Yaskawa INFORM job: A_ROOF_UPPER_0614_2_PAINT_18.JBI

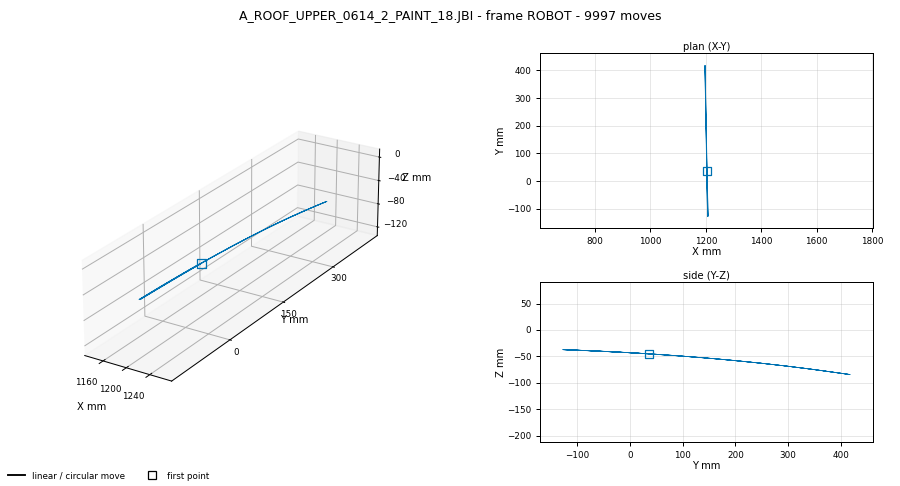
[picture p0: tool path of A_ROOF_UPPER_0614_2_PAINT_18.JBI in frame ROBOT, 9997 of 9997 moves have a stored position in this frame; points joined in program order, loops and branches not executed]
/JOB
//NAME A_ROOF_UPPER_0614_2_PAINT18
//POS
///NPOS 9997,0,0,0,0,0
///TOOL 1
///USER 0
///POSTYPE ROBOT
///RECTAN
///RCONF 1,0,0,0,0,0,0,0,0,0,0,0,0,0,0,0,0,0,0,0,0,0,0,0
C00000=1205.007,36.584,-45.184,-179.345,5.640,148.798
C00001=1205.012,36.335,-45.168,-179.348,5.639,148.799
C00002=1205.017,36.086,-45.153,-179.350,5.639,148.800
C00003=1205.023,35.836,-45.137,-179.353,5.638,148.800
C00004=1205.027,35.586,-45.122,-179.356,5.638,148.801
C00005=1205.032,35.337,-45.106,-179.358,5.637,148.801
C00006=1205.037,35.088,-45.090,-179.360,5.636,148.802
C00007=1205.042,34.839,-45.075,-179.363,5.636,148.803
C00008=1205.047,34.589,-45.059,-179.366,5.635,148.803
C00009=1205.052,34.340,-45.043,-179.368,5.635,148.804
C00010=1205.057,34.090,-45.028,-179.371,5.634,148.805
C00011=1205.062,33.841,-45.013,-179.373,5.633,148.805
C00012=1205.067,33.591,-44.997,-179.376,5.633,148.806
C00013=1205.072,33.342,-44.982,-179.378,5.632,148.807
C00014=1205.077,33.093,-44.966,-179.381,5.632,148.807
C00015=1205.082,32.843,-44.951,-179.383,5.631,148.808
C00016=1205.086,32.593,-44.935,-179.386,5.630,148.808
C00017=1205.092,32.344,-44.920,-179.389,5.630,148.809
C00018=1205.097,32.094,-44.905,-179.391,5.629,148.810
C00019=1205.102,31.845,-44.890,-179.394,5.629,148.810
C00020=1205.107,31.595,-44.874,-179.396,5.628,148.811
C00021=1205.112,31.345,-44.858,-179.399,5.627,148.811
C00022=1205.117,31.096,-44.843,-179.401,5.627,148.812
C00023=1205.122,30.847,-44.828,-179.404,5.626,148.813
C00024=1205.127,30.598,-44.813,-179.407,5.626,148.814
C00025=1205.132,30.348,-44.797,-179.409,5.625,148.814
C00026=1205.137,30.098,-44.781,-179.411,5.624,148.815
C00027=1205.142,29.849,-44.766,-179.414,5.624,148.815
C00028=1205.147,29.600,-44.750,-179.417,5.623,148.816
C00029=1205.152,29.331,-44.735,-179.419,5.623,148.817
C00030=1205.158,29.062,-44.718,-179.422,5.622,148.817
C00031=1205.164,28.793,-44.701,-179.425,5.622,148.818
C00032=1205.169,28.525,-44.686,-179.427,5.621,148.819
C00033=1205.174,28.274,-44.670,-179.430,5.621,148.819
C00034=1205.178,28.025,-44.655,-179.432,5.620,148.820
C00035=1205.184,27.776,-44.639,-179.435,5.619,148.821
C00036=1205.188,27.527,-44.624,-179.437,5.619,148.821
C00037=1205.194,27.277,-44.609,-179.440,5.618,148.822
C00038=1205.199,27.028,-44.594,-179.443,5.618,148.823
C00039=1205.204,26.778,-44.579,-179.445,5.617,148.823
C00040=1205.208,26.529,-44.563,-179.447,5.616,148.824
C00041=1205.213,26.279,-44.548,-179.450,5.616,148.824
C00042=1205.218,26.029,-44.534,-179.453,5.615,148.825
C00043=1205.224,25.780,-44.518,-179.455,5.615,148.826
C00044=1205.228,25.531,-44.503,-179.458,5.614,148.826
C00045=1205.234,25.282,-44.487,-179.460,5.613,148.827
C00046=1205.239,25.032,-44.473,-179.463,5.613,148.828
C00047=1205.244,24.782,-44.457,-179.465,5.612,148.828
C00048=1205.248,24.533,-44.442,-179.468,5.612,148.829
C00049=1205.253,24.283,-44.428,-179.471,5.611,148.830
C00050=1205.259,24.034,-44.412,-179.473,5.610,148.830
C00051=1205.263,23.784,-44.397,-179.476,5.610,148.831
C00052=1205.269,23.534,-44.382,-179.478,5.609,148.831
C00053=1205.274,23.285,-44.367,-179.481,5.609,148.832
C00054=1205.279,23.036,-44.352,-179.483,5.608,148.833
C00055=1205.284,22.786,-44.338,-179.486,5.608,148.833
C00056=1205.289,22.537,-44.323,-179.488,5.607,148.834
C00057=1205.294,22.288,-44.307,-179.490,5.607,148.835
C00058=1205.299,22.038,-44.293,-179.493,5.607,148.835
C00059=1205.304,21.789,-44.277,-179.496,5.606,148.836
C00060=1205.309,21.538,-44.262,-179.498,5.606,148.837
C00061=1205.313,21.289,-44.247,-179.501,5.605,148.837
C00062=1205.319,21.040,-44.232,-179.503,5.604,148.838
C00063=1205.324,20.790,-44.218,-179.506,5.604,148.838
C00064=1205.328,20.541,-44.203,-179.508,5.603,148.839
C00065=1205.334,20.291,-44.188,-179.511,5.603,148.840
C00066=1205.339,20.042,-44.173,-179.514,5.602,148.840
C00067=1205.344,19.792,-44.158,-179.516,5.601,148.841
C00068=1205.349,19.543,-44.143,-179.519,5.601,148.842
C00069=1205.354,19.293,-44.129,-179.521,5.600,148.842
C00070=1205.359,19.044,-44.114,-179.524,5.600,148.843
C00071=1205.364,18.794,-44.099,-179.526,5.599,148.844
C00072=1205.369,18.545,-44.084,-179.529,5.599,148.844
C00073=1205.374,18.295,-44.069,-179.531,5.599,148.845
C00074=1205.379,18.046,-44.054,-179.533,5.598,148.845
C00075=1205.384,17.796,-44.040,-179.536,5.598,148.846
C00076=1205.389,17.547,-44.025,-179.539,5.597,148.847
C00077=1205.395,17.297,-44.010,-179.541,5.597,148.847
C00078=1205.399,17.048,-43.995,-179.544,5.596,148.848
C00079=1205.404,16.798,-43.980,-179.546,5.595,148.849
C00080=1205.409,16.549,-43.965,-179.549,5.595,148.849
C00081=1205.414,16.299,-43.951,-179.551,5.594,148.850
C00082=1205.419,16.049,-43.936,-179.554,5.594,148.851
C00083=1205.424,15.800,-43.921,-179.557,5.593,148.851
C00084=1205.429,15.550,-43.907,-179.559,5.593,148.852
C00085=1205.434,15.301,-43.891,-179.561,5.592,148.852
C00086=1205.439,15.051,-43.877,-179.564,5.592,148.853
C00087=1205.444,14.802,-43.863,-179.566,5.592,148.854
C00088=1205.449,14.552,-43.848,-179.569,5.591,148.855
C00089=1205.455,14.302,-43.833,-179.571,5.591,148.855
C00090=1205.460,14.053,-43.819,-179.574,5.590,148.856
C00091=1205.464,13.804,-43.804,-179.576,5.589,148.856
C00092=1205.469,13.554,-43.789,-179.579,5.589,148.857
C00093=1205.475,13.305,-43.776,-179.582,5.588,148.858
C00094=1205.480,13.056,-43.760,-179.584,5.588,148.858
C00095=1205.485,12.806,-43.746,-179.587,5.587,148.859
C00096=1205.490,12.556,-43.731,-179.589,5.588,148.860
C00097=1205.495,12.307,-43.716,-179.592,5.587,148.860
C00098=1205.500,12.057,-43.702,-179.594,5.586,148.861
C00099=1205.505,11.808,-43.688,-179.596,5.586,148.862
C00100=1205.510,11.558,-43.672,-179.599,5.585,148.862
C00101=1205.515,11.308,-43.658,-179.602,5.585,148.863
C00102=1205.520,11.059,-43.644,-179.604,5.584,148.864
C00103=1205.525,10.809,-43.629,-179.607,5.584,148.864
C00104=1205.530,10.561,-43.615,-179.609,5.583,148.865
C00105=1205.535,10.311,-43.601,-179.612,5.582,148.865
C00106=1205.540,10.061,-43.586,-179.614,5.583,148.866
C00107=1205.545,9.812,-43.572,-179.617,5.582,148.867
C00108=1205.551,9.562,-43.557,-179.619,5.582,148.868
C00109=1205.555,9.312,-43.542,-179.622,5.581,148.868
C00110=1205.560,9.063,-43.528,-179.624,5.580,148.869
C00111=1205.565,8.813,-43.514,-179.627,5.580,148.869
C00112=1205.570,8.563,-43.499,-179.629,5.579,148.870
C00113=1205.576,8.314,-43.485,-179.632,5.579,148.871
C00114=1205.581,8.065,-43.471,-179.635,5.578,148.871
C00115=1205.585,7.815,-43.456,-179.637,5.578,148.872
C00116=1205.590,7.566,-43.442,-179.639,5.578,148.873
C00117=1205.595,7.316,-43.428,-179.642,5.577,148.873
C00118=1205.600,7.066,-43.413,-179.644,5.577,148.874
C00119=1205.606,6.817,-43.399,-179.647,5.576,148.875
C00120=1205.611,6.568,-43.385,-179.649,5.576,148.875
C00121=1205.616,6.318,-43.371,-179.652,5.575,148.876
C00122=1205.621,6.068,-43.357,-179.655,5.575,148.877
C00123=1205.625,5.819,-43.342,-179.657,5.575,148.877
C00124=1205.630,5.569,-43.327,-179.659,5.574,148.878
C00125=1205.636,5.320,-43.313,-179.662,5.573,148.879
C00126=1205.641,5.071,-43.299,-179.664,5.573,148.879
C00127=1205.646,4.821,-43.285,-179.667,5.572,148.880
C00128=1205.651,4.571,-43.271,-179.670,5.572,148.881
C00129=1205.656,4.322,-43.256,-179.672,5.571,148.881
C00130=1205.661,4.073,-43.242,-179.675,5.571,148.882
C00131=1205.666,3.823,-43.228,-179.677,5.571,148.882
C00132=1205.671,3.573,-43.214,-179.679,5.570,148.883
C00133=1205.677,3.304,-43.199,-179.682,5.570,148.884
C00134=1205.682,3.035,-43.183,-179.684,5.569,148.884
C00135=1205.687,2.766,-43.168,-179.687,5.569,148.885
C00136=1205.694,2.497,-43.152,-179.690,5.569,148.886
C00137=1205.698,2.248,-43.139,-179.692,5.568,148.887
C00138=1205.703,1.998,-43.124,-179.695,5.567,148.887
C00139=1205.708,1.748,-43.110,-179.698,5.567,148.888
C00140=1205.714,1.499,-43.097,-179.700,5.566,148.889
C00141=1205.718,1.249,-43.082,-179.703,5.566,148.889
C00142=1205.723,0.999,-43.068,-179.705,5.566,148.890
C00143=1205.728,0.750,-43.054,-179.708,5.566,148.891
C00144=1205.734,0.501,-43.040,-179.710,5.565,148.891
C00145=1205.739,0.251,-43.026,-179.713,5.564,148.892
C00146=1205.744,0.001,-43.011,-179.715,5.564,148.893
C00147=1205.749,-0.249,-42.997,-179.718,5.563,148.893
C00148=1205.754,-0.497,-42.984,-179.720,5.564,148.894
C00149=1205.759,-0.747,-42.970,-179.723,5.563,148.895
C00150=1205.764,-0.997,-42.956,-179.725,5.563,148.895
C00151=1205.769,-1.247,-42.942,-179.727,5.562,148.896
C00152=1205.774,-1.496,-42.928,-179.730,5.561,148.896
C00153=1205.779,-1.746,-42.914,-179.733,5.561,148.897
C00154=1205.784,-1.995,-42.899,-179.735,5.561,148.898
C00155=1205.789,-2.244,-42.886,-179.737,5.561,148.898
C00156=1205.794,-2.494,-42.872,-179.740,5.560,148.899
C00157=1205.799,-2.744,-42.858,-179.743,5.560,148.900
C00158=1205.805,-2.993,-42.844,-179.745,5.559,148.901
C00159=1205.810,-3.243,-42.830,-179.748,5.558,148.901
C00160=1205.815,-3.493,-42.816,-179.750,5.559,148.902
C00161=1205.820,-3.742,-42.803,-179.752,5.558,148.902
C00162=1205.825,-3.992,-42.789,-179.755,5.558,148.903
C00163=1205.830,-4.241,-42.775,-179.758,5.557,148.904
C00164=1205.835,-4.491,-42.760,-179.760,5.557,148.904
C00165=1205.840,-4.740,-42.746,-179.763,5.556,148.905
C00166=1205.845,-4.990,-42.733,-179.765,5.556,148.906
C00167=1205.850,-5.239,-42.719,-179.767,5.556,148.906
C00168=1205.855,-5.489,-42.705,-179.770,5.555,148.907
C00169=1205.861,-5.739,-42.692,-179.772,5.555,148.908
C00170=1205.865,-5.988,-42.678,-179.775,5.554,148.908
C00171=1205.870,-6.238,-42.664,-179.778,5.554,148.909
C00172=1205.875,-6.487,-42.650,-179.780,5.554,148.910
C00173=1205.881,-6.737,-42.637,-179.783,5.553,148.910
C00174=1205.885,-6.986,-42.623,-179.785,5.552,148.911
C00175=1205.890,-7.236,-42.609,-179.787,5.552,148.912
C00176=1205.896,-7.486,-42.595,-179.790,5.552,148.912
C00177=1205.900,-7.735,-42.582,-179.792,5.552,148.913
C00178=1205.905,-7.985,-42.567,-179.795,5.551,148.914
C00179=1205.911,-8.234,-42.554,-179.797,5.551,148.914
C00180=1205.916,-8.484,-42.540,-179.800,5.550,148.915
C00181=1205.921,-8.733,-42.527,-179.803,5.550,148.916
C00182=1205.926,-8.983,-42.513,-179.805,5.549,148.916
C00183=1205.931,-9.233,-42.499,-179.807,5.549,148.917
C00184=1205.936,-9.482,-42.486,-179.810,5.549,148.918
C00185=1205.941,-9.732,-42.472,-179.812,5.548,148.918
C00186=1205.947,-9.982,-42.459,-179.815,5.548,148.919
C00187=1205.951,-10.231,-42.445,-179.818,5.547,148.920
C00188=1205.956,-10.481,-42.431,-179.820,5.548,148.920
C00189=1205.962,-10.730,-42.418,-179.822,5.547,148.921
C00190=1205.966,-10.980,-42.404,-179.824,5.546,148.922
C00191=1205.972,-11.229,-42.391,-179.827,5.546,148.922
C00192=1205.977,-11.479,-42.377,-179.830,5.545,148.923
C00193=1205.982,-11.728,-42.364,-179.832,5.546,148.924
C00194=1205.987,-11.978,-42.350,-179.835,5.545,148.924
C00195=1205.992,-12.228,-42.337,-179.837,5.545,148.925
C00196=1205.997,-12.477,-42.323,-179.840,5.544,148.926
C00197=1206.002,-12.727,-42.310,-179.842,5.544,148.926
C00198=1206.007,-12.976,-42.296,-179.844,5.544,148.927
C00199=1206.013,-13.226,-42.282,-179.847,5.543,148.928
C00200=1206.018,-13.475,-42.269,-179.849,5.543,148.928
C00201=1206.023,-13.725,-42.255,-179.852,5.542,148.929
C00202=1206.028,-13.974,-42.242,-179.854,5.543,148.930
C00203=1206.033,-14.224,-42.228,-179.857,5.542,148.930
C00204=1206.038,-14.473,-42.215,-179.859,5.542,148.931
C00205=1206.043,-14.723,-42.202,-179.862,5.541,148.932
C00206=1206.049,-14.973,-42.188,-179.864,5.540,148.932
C00207=1206.053,-15.223,-42.175,-179.866,5.541,148.933
C00208=1206.059,-15.472,-42.162,-179.869,5.540,148.934
C00209=1206.063,-15.722,-42.148,-179.872,5.540,148.934
C00210=1206.069,-15.971,-42.135,-179.874,5.539,148.935
C00211=1206.073,-16.221,-42.121,-179.877,5.539,148.936
C00212=1206.079,-16.470,-42.108,-179.879,5.539,148.936
C00213=1206.084,-16.720,-42.095,-179.882,5.538,148.937
C00214=1206.089,-16.969,-42.081,-179.884,5.538,148.937
C00215=1206.094,-17.219,-42.068,-179.887,5.537,148.938
C00216=1206.100,-17.469,-42.055,-179.889,5.537,148.939
C00217=1206.104,-17.718,-42.041,-179.891,5.537,148.940
C00218=1206.110,-17.968,-42.028,-179.894,5.536,148.940
C00219=1206.114,-18.218,-42.015,-179.897,5.536,148.941
C00220=1206.120,-18.467,-42.001,-179.899,5.536,148.942
C00221=1206.124,-18.717,-41.988,-179.901,5.536,148.942
C00222=1206.130,-18.967,-41.975,-179.903,5.535,148.943
C00223=1206.134,-19.216,-41.961,-179.906,5.534,148.943
C00224=1206.140,-19.466,-41.948,-179.909,5.534,148.944
C00225=1206.145,-19.715,-41.935,-179.911,5.534,148.945
C00226=1206.151,-19.965,-41.922,-179.914,5.534,148.946
C00227=1206.155,-20.214,-41.908,-179.916,5.533,148.946
C00228=1206.161,-20.464,-41.895,-179.919,5.533,148.947
C00229=1206.166,-20.714,-41.882,-179.921,5.533,148.948
C00230=1206.170,-20.964,-41.869,-179.923,5.532,148.948
C00231=1206.176,-21.213,-41.855,-179.926,5.532,148.949
C00232=1206.181,-21.462,-41.843,-179.928,5.531,148.950
C00233=1206.186,-21.712,-41.829,-179.930,5.532,148.950
C00234=1206.191,-21.962,-41.817,-179.933,5.531,148.951
C00235=1206.196,-22.212,-41.804,-179.936,5.531,148.952
C00236=1206.201,-22.461,-41.790,-179.938,5.530,148.952
C00237=1206.206,-22.730,-41.776,-179.941,5.530,148.953
C00238=1206.212,-23.000,-41.762,-179.943,5.530,148.954
C00239=1206.218,-23.269,-41.747,-179.946,5.530,148.954
C00240=1206.223,-23.539,-41.733,-179.949,5.529,148.955
C00241=1206.229,-23.788,-41.720,-179.951,5.529,148.956
C00242=1206.234,-24.038,-41.707,-179.954,5.528,148.956
C00243=1206.239,-24.288,-41.695,-179.956,5.528,148.957
C00244=1206.244,-24.537,-41.681,-179.959,5.528,148.958
C00245=1206.249,-24.787,-41.668,-179.961,5.528,148.959
C00246=1206.254,-25.036,-41.655,-179.963,5.527,148.959
C00247=1206.259,-25.286,-41.642,-179.966,5.527,148.960
C00248=1206.264,-25.536,-41.629,-179.968,5.527,148.960
C00249=1206.269,-25.785,-41.616,-179.971,5.526,148.961
C00250=1206.274,-26.035,-41.604,-179.973,5.526,148.962
C00251=1206.280,-26.285,-41.590,-179.976,5.526,148.963
C00252=1206.285,-26.534,-41.578,-179.978,5.525,148.963
C00253=1206.289,-26.784,-41.565,-179.981,5.525,148.964
C00254=1206.295,-27.034,-41.552,-179.984,5.524,148.965
C00255=1206.300,-27.283,-41.539,-179.985,5.524,148.965
C00256=1206.305,-27.532,-41.525,-179.988,5.524,148.966
C00257=1206.310,-27.782,-41.513,-179.990,5.523,148.966
C00258=1206.316,-28.031,-41.499,-179.993,5.523,148.967
C00259=1206.320,-28.281,-41.487,-179.995,5.523,148.968
C00260=1206.325,-28.531,-41.474,-179.998,5.523,148.969
C00261=1206.331,-28.780,-41.461,179.999,5.522,148.969
C00262=1206.336,-29.030,-41.448,179.997,5.523,148.970
C00263=1206.341,-29.280,-41.435,179.995,5.522,148.970
C00264=1206.346,-29.529,-41.423,179.993,5.521,148.971
C00265=1206.350,-29.779,-41.410,179.990,5.521,148.972
C00266=1206.356,-30.029,-41.396,179.988,5.521,148.973
C00267=1206.361,-30.278,-41.384,179.985,5.521,148.973
C00268=1206.366,-30.529,-41.372,179.982,5.520,148.974
C00269=1206.371,-30.778,-41.359,179.980,5.520,148.975
C00270=1206.377,-31.028,-41.346,179.978,5.520,148.975
C00271=1206.382,-31.277,-41.333,179.975,5.520,148.976
C00272=1206.387,-31.527,-41.320,179.973,5.519,148.976
C00273=1206.392,-31.776,-41.308,179.971,5.519,148.977
C00274=1206.397,-32.026,-41.295,179.968,5.519,148.978
C00275=1206.402,-32.275,-41.282,179.966,5.518,148.979
C00276=1206.408,-32.525,-41.269,179.963,5.518,148.979
C00277=1206.413,-32.774,-41.256,179.961,5.518,148.980
C00278=1206.418,-33.024,-41.244,179.958,5.518,148.981
C00279=1206.423,-33.274,-41.232,179.955,5.517,148.981
C00280=1206.428,-33.524,-41.219,179.954,5.517,148.982
C00281=1206.433,-33.773,-41.206,179.951,5.517,148.983
C00282=1206.439,-34.023,-41.193,179.949,5.516,148.983
C00283=1206.444,-34.272,-41.180,179.946,5.516,148.984
C00284=1206.448,-34.522,-41.167,179.944,5.516,148.985
C00285=1206.454,-34.772,-41.156,179.941,5.516,148.985
C00286=1206.459,-35.021,-41.143,179.938,5.515,148.986
C00287=1206.464,-35.271,-41.130,179.936,5.515,148.987
C00288=1206.469,-35.521,-41.117,179.934,5.515,148.987
C00289=1206.474,-35.770,-41.105,179.932,5.514,148.988
C00290=1206.480,-36.020,-41.092,179.929,5.514,148.989
C00291=1206.485,-36.270,-41.080,179.927,5.514,148.989
C00292=1206.490,-36.519,-41.067,179.924,5.514,148.990
C00293=1206.495,-36.769,-41.054,179.921,5.513,148.991
C00294=1206.500,-37.018,-41.041,179.919,5.513,148.991
C00295=1206.505,-37.268,-41.030,179.917,5.513,148.992
C00296=1206.510,-37.517,-41.017,179.914,5.512,148.993
C00297=1206.515,-37.767,-41.004,179.913,5.512,148.993
C00298=1206.520,-38.017,-40.992,179.910,5.512,148.994
C00299=1206.525,-38.267,-40.980,179.907,5.511,148.995
C00300=1206.530,-38.516,-40.967,179.905,5.512,148.995
C00301=1206.536,-38.765,-40.954,179.902,5.511,148.996
C00302=1206.541,-39.015,-40.942,179.900,5.511,148.997
C00303=1206.546,-39.265,-40.930,179.897,5.510,148.997
C00304=1206.551,-39.515,-40.917,179.895,5.511,148.998
C00305=1206.556,-39.765,-40.905,179.892,5.510,148.999
C00306=1206.561,-40.014,-40.892,179.890,5.509,148.999
C00307=1206.566,-40.263,-40.880,179.888,5.510,149.000
C00308=1206.572,-40.513,-40.868,179.885,5.509,149.001
C00309=1206.577,-40.762,-40.855,179.883,5.509,149.001
C00310=1206.582,-41.012,-40.843,179.881,5.509,149.002
C00311=1206.587,-41.262,-40.830,179.878,5.509,149.003
C00312=1206.592,-41.512,-40.818,179.875,5.508,149.004
C00313=1206.597,-41.762,-40.806,179.873,5.509,149.004
C00314=1206.603,-42.011,-40.793,179.871,5.508,149.005
C00315=1206.608,-42.260,-40.781,179.868,5.507,149.005
C00316=1206.613,-42.510,-40.769,179.866,5.508,149.006
C00317=1206.618,-42.760,-40.756,179.864,5.507,149.007
C00318=1206.624,-43.009,-40.744,179.861,5.507,149.008
C00319=1206.628,-43.259,-40.731,179.859,5.507,149.008
C00320=1206.633,-43.509,-40.719,179.856,5.507,149.009
C00321=1206.639,-43.759,-40.707,179.854,5.506,149.010
C00322=1206.644,-44.008,-40.694,179.852,5.506,149.010
C00323=1206.649,-44.258,-40.682,179.849,5.506,149.011
C00324=1206.654,-44.507,-40.670,179.847,5.505,149.011
C00325=1206.660,-44.757,-40.658,179.845,5.506,149.012
C00326=1206.665,-45.007,-40.645,179.842,5.505,149.013
C00327=1206.670,-45.256,-40.634,179.839,5.505,149.014
C00328=1206.675,-45.505,-40.621,179.837,5.504,149.014
C00329=1206.680,-45.755,-40.610,179.835,5.505,149.015
C00330=1206.685,-46.005,-40.597,179.832,5.504,149.015
C00331=1206.690,-46.255,-40.585,179.830,5.503,149.016
C00332=1206.695,-46.505,-40.572,179.828,5.504,149.017
C00333=1206.701,-46.755,-40.560,179.825,5.503,149.018
C00334=1206.706,-47.004,-40.548,179.822,5.503,149.018
C00335=1206.711,-47.254,-40.536,179.820,5.503,149.019
C00336=1206.716,-47.503,-40.524,179.818,5.503,149.020
C00337=1206.721,-47.753,-40.512,179.815,5.503,149.020
C00338=1206.727,-48.003,-40.500,179.813,5.502,149.021
C00339=1206.732,-48.252,-40.487,179.811,5.502,149.022
C00340=1206.737,-48.502,-40.476,179.809,5.502,149.022
C00341=1206.742,-48.772,-40.463,179.806,5.501,149.023
C00342=1206.748,-49.041,-40.449,179.803,5.501,149.024
C00343=1206.753,-49.312,-40.436,179.800,5.501,149.025
C00344=1206.759,-49.582,-40.423,179.797,5.500,149.025
C00345=1206.764,-49.832,-40.411,179.795,5.501,149.026
C00346=1206.769,-50.081,-40.399,179.793,5.500,149.026
C00347=1206.775,-50.331,-40.387,179.790,5.500,149.027
C00348=1206.780,-50.581,-40.375,179.788,5.500,149.028
C00349=1206.784,-50.830,-40.363,179.786,5.499,149.029
C00350=1206.790,-51.080,-40.351,179.783,5.499,149.029
C00351=1206.795,-51.330,-40.339,179.781,5.499,149.030
C00352=1206.800,-51.579,-40.327,179.778,5.499,149.031
C00353=1206.805,-51.829,-40.315,179.777,5.499,149.031
C00354=1206.810,-52.079,-40.304,179.774,5.498,149.032
C00355=1206.816,-52.328,-40.291,179.771,5.498,149.033
C00356=1206.821,-52.578,-40.279,179.769,5.498,149.033
C00357=1206.826,-52.828,-40.268,179.767,5.498,149.034
C00358=1206.831,-53.077,-40.255,179.764,5.497,149.035
C00359=1206.836,-53.327,-40.243,179.762,5.498,149.035
C00360=1206.842,-53.577,-40.231,179.759,5.497,149.036
C00361=1206.847,-53.826,-40.220,179.757,5.496,149.037
C00362=1206.852,-54.075,-40.208,179.755,5.497,149.037
C00363=1206.858,-54.325,-40.196,179.752,5.496,149.038
C00364=1206.862,-54.575,-40.185,179.750,5.496,149.039
C00365=1206.868,-54.825,-40.173,179.748,5.496,149.039
C00366=1206.873,-55.074,-40.160,179.745,5.496,149.040
C00367=1206.878,-55.324,-40.149,179.743,5.496,149.041
C00368=1206.883,-55.574,-40.137,179.740,5.496,149.042
C00369=1206.888,-55.824,-40.125,179.738,5.495,149.042
C00370=1206.893,-56.073,-40.114,179.736,5.495,149.043
C00371=1206.898,-56.323,-40.101,179.733,5.495,149.043
C00372=1206.904,-56.573,-40.089,179.731,5.494,149.044
C00373=1206.908,-56.822,-40.078,179.728,5.495,149.045
C00374=1206.914,-57.072,-40.066,179.726,5.494,149.046
C00375=1206.919,-57.322,-40.054,179.723,5.494,149.046
C00376=1206.924,-57.572,-40.043,179.721,5.494,149.047
C00377=1206.929,-57.821,-40.030,179.719,5.493,149.047
C00378=1206.935,-58.070,-40.019,179.717,5.494,149.048
C00379=1206.940,-58.320,-40.008,179.714,5.493,149.049
C00380=1206.945,-58.570,-39.996,179.711,5.493,149.050
C00381=1206.950,-58.819,-39.984,179.709,5.493,149.050
C00382=1206.955,-59.069,-39.973,179.707,5.493,149.051
C00383=1206.961,-59.319,-39.961,179.704,5.492,149.052
C00384=1206.965,-59.569,-39.949,179.702,5.492,149.052
C00385=1206.971,-59.819,-39.937,179.700,5.492,149.053
C00386=1206.975,-60.068,-39.925,179.698,5.492,149.054
C00387=1206.981,-60.317,-39.914,179.695,5.492,149.054
C00388=1206.987,-60.567,-39.902,179.692,5.491,149.055
C00389=1206.991,-60.817,-39.891,179.690,5.491,149.056
C00390=1206.997,-61.067,-39.879,179.688,5.491,149.056
C00391=1207.001,-61.316,-39.868,179.686,5.491,149.057
C00392=1207.007,-61.566,-39.856,179.683,5.491,149.058
C00393=1207.012,-61.816,-39.844,179.681,5.490,149.058
C00394=1207.018,-62.065,-39.833,179.679,5.490,149.059
C00395=1207.022,-62.315,-39.822,179.676,5.490,149.060
C00396=1207.028,-62.565,-39.810,179.673,5.490,149.060
C00397=1207.033,-62.814,-39.798,179.671,5.490,149.061
C00398=1207.038,-63.064,-39.787,179.669,5.489,149.062
C00399=1207.043,-63.314,-39.775,179.667,5.489,149.062
C00400=1207.048,-63.564,-39.763,179.664,5.489,149.063
C00401=1207.054,-63.813,-39.752,179.662,5.489,149.064
C00402=1207.059,-64.063,-39.741,179.659,5.489,149.064
C00403=1207.064,-64.312,-39.729,179.657,5.488,149.065
C00404=1207.069,-64.562,-39.717,179.655,5.489,149.066
C00405=1207.074,-64.812,-39.705,179.653,5.488,149.066
C00406=1207.080,-65.061,-39.695,179.650,5.488,149.067
C00407=1207.085,-65.311,-39.683,179.648,5.488,149.068
C00408=1207.090,-65.561,-39.671,179.645,5.487,149.068
C00409=1207.095,-65.811,-39.660,179.643,5.488,149.069
C00410=1207.100,-66.061,-39.649,179.640,5.487,149.070
C00411=1207.106,-66.310,-39.637,179.638,5.487,149.070
C00412=1207.111,-66.560,-39.626,179.636,5.487,149.071
C00413=1207.116,-66.809,-39.615,179.633,5.486,149.072
C00414=1207.121,-67.059,-39.603,179.631,5.487,149.072
C00415=1207.126,-67.309,-39.592,179.629,5.486,149.073
C00416=1207.132,-67.558,-39.580,179.626,5.486,149.074
C00417=1207.137,-67.808,-39.570,179.624,5.486,149.074
C00418=1207.142,-68.058,-39.558,179.622,5.485,149.075
C00419=1207.147,-68.308,-39.546,179.620,5.486,149.076
C00420=1207.152,-68.557,-39.535,179.617,5.485,149.076
C00421=1207.157,-68.807,-39.524,179.614,5.485,149.077
C00422=1207.162,-69.056,-39.512,179.612,5.485,149.078
C00423=1207.168,-69.307,-39.501,179.610,5.485,149.078
C00424=1207.173,-69.556,-39.490,179.607,5.485,149.079
C00425=1207.179,-69.806,-39.478,179.605,5.484,149.080
C00426=1207.183,-70.055,-39.467,179.603,5.484,149.080
C00427=1207.188,-70.305,-39.456,179.601,5.484,149.081
C00428=1207.194,-70.555,-39.445,179.598,5.484,149.082
C00429=1207.199,-70.804,-39.434,179.596,5.484,149.082
C00430=1207.204,-71.054,-39.422,179.593,5.484,149.083
C00431=1207.210,-71.303,-39.411,179.591,5.483,149.084
C00432=1207.215,-71.554,-39.400,179.589,5.483,149.084
C00433=1207.220,-71.803,-39.388,179.586,5.483,149.085
C00434=1207.225,-72.053,-39.377,179.584,5.483,149.086
C00435=1207.230,-72.302,-39.366,179.581,5.483,149.087
C00436=1207.236,-72.553,-39.355,179.579,5.483,149.087
C00437=1207.241,-72.802,-39.344,179.577,5.482,149.088
C00438=1207.246,-73.051,-39.333,179.574,5.482,149.088
C00439=1207.251,-73.301,-39.321,179.572,5.482,149.089
C00440=1207.256,-73.551,-39.310,179.570,5.482,149.090
C00441=1207.262,-73.800,-39.299,179.568,5.482,149.091
C00442=1207.267,-74.050,-39.287,179.565,5.482,149.091
C00443=1207.272,-74.300,-39.277,179.562,5.481,149.092
C00444=1207.277,-74.549,-39.266,179.561,5.481,149.092
C00445=1207.283,-74.820,-39.254,179.558,5.481,149.093
C00446=1207.289,-75.091,-39.241,179.555,5.481,149.094
C00447=1207.294,-75.361,-39.230,179.553,5.481,149.095
C00448=1207.300,-75.632,-39.218,179.550,5.481,149.096
C00449=1207.305,-75.882,-39.206,179.548,5.480,149.096
C00450=1207.311,-76.132,-39.196,179.546,5.480,149.097
C00451=1207.315,-76.381,-39.185,179.543,5.480,149.097
C00452=1207.320,-76.631,-39.173,179.541,5.480,149.098
C00453=1207.326,-76.881,-39.162,179.538,5.480,149.099
C00454=1207.331,-77.130,-39.151,179.536,5.480,149.100
C00455=1207.336,-77.381,-39.141,179.534,5.479,149.100
C00456=1207.341,-77.630,-39.130,179.532,5.480,149.101
C00457=1207.347,-77.880,-39.119,179.529,5.479,149.101
C00458=1207.352,-78.129,-39.108,179.527,5.479,149.102
C00459=1207.357,-78.379,-39.096,179.525,5.479,149.103
C00460=1207.362,-78.629,-39.086,179.522,5.479,149.104
C00461=1207.367,-78.878,-39.075,179.520,5.479,149.104
C00462=1207.373,-79.128,-39.064,179.518,5.478,149.105
C00463=1207.378,-79.378,-39.052,179.516,5.479,149.105
C00464=1207.383,-79.628,-39.042,179.513,5.478,149.106
C00465=1207.388,-79.877,-39.031,179.510,5.478,149.107
C00466=1207.394,-80.127,-39.021,179.508,5.478,149.108
C00467=1207.399,-80.377,-39.009,179.506,5.477,149.108
C00468=1207.404,-80.627,-38.998,179.504,5.478,149.109
C00469=1207.409,-80.876,-38.987,179.501,5.477,149.109
C00470=1207.414,-81.126,-38.977,179.499,5.478,149.110
C00471=1207.420,-81.375,-38.966,179.496,5.477,149.111
C00472=1207.425,-81.625,-38.955,179.494,5.478,149.112
C00473=1207.431,-81.875,-38.944,179.492,5.477,149.112
C00474=1207.436,-82.125,-38.933,179.489,5.476,149.113
C00475=1207.440,-82.374,-38.922,179.487,5.477,149.113
C00476=1207.446,-82.624,-38.912,179.485,5.476,149.114
C00477=1207.451,-82.874,-38.901,179.483,5.477,149.115
C00478=1207.456,-83.123,-38.890,179.480,5.476,149.115
C00479=1207.461,-83.373,-38.880,179.478,5.476,149.116
C00480=1207.467,-83.622,-38.869,179.476,5.476,149.117
C00481=1207.472,-83.873,-38.857,179.474,5.476,149.118
C00482=1207.477,-84.122,-38.846,179.471,5.476,149.118
C00483=1207.483,-84.372,-38.836,179.469,5.475,149.119
C00484=1207.488,-84.622,-38.825,179.467,5.475,149.119
C00485=1207.493,-84.871,-38.814,179.464,5.475,149.120
C00486=1207.498,-85.121,-38.804,179.462,5.475,149.121
C00487=1207.504,-85.371,-38.794,179.459,5.475,149.122
C00488=1207.508,-85.621,-38.782,179.457,5.475,149.122
C00489=1207.514,-85.870,-38.772,179.455,5.474,149.123
C00490=1207.519,-86.120,-38.761,179.453,5.475,149.123
C00491=1207.524,-86.369,-38.751,179.450,5.474,149.124
C00492=1207.529,-86.620,-38.740,179.448,5.474,149.125
C00493=1207.534,-86.868,-38.729,179.445,5.474,149.126
C00494=1207.539,-87.119,-38.719,179.443,5.473,149.126
C00495=1207.545,-87.368,-38.708,179.441,5.474,149.127
C00496=1207.550,-87.619,-38.698,179.439,5.473,149.127
C00497=1207.556,-87.868,-38.686,179.436,5.474,149.128
C00498=1207.561,-88.118,-38.676,179.434,5.473,149.129
C00499=1207.567,-88.368,-38.665,179.432,5.473,149.129
C00500=1207.571,-88.617,-38.654,179.429,5.473,149.130
C00501=1207.577,-88.867,-38.644,179.427,5.473,149.131
C00502=1207.582,-89.117,-38.633,179.425,5.473,149.132
C00503=1207.588,-89.366,-38.623,179.423,5.473,149.132
C00504=1207.592,-89.616,-38.612,179.420,5.472,149.133
C00505=1207.598,-89.866,-38.602,179.418,5.472,149.133
C00506=1207.603,-90.116,-38.591,179.416,5.472,149.134
C00507=1207.608,-90.365,-38.581,179.413,5.472,149.135
C00508=1207.612,-90.615,-38.570,179.411,5.472,149.136
C00509=1207.618,-90.864,-38.560,179.409,5.471,149.136
C00510=1207.623,-91.115,-38.549,179.407,5.472,149.137
C00511=1207.629,-91.364,-38.539,179.404,5.471,149.137
C00512=1207.634,-91.614,-38.529,179.402,5.472,149.138
C00513=1207.639,-91.863,-38.518,179.399,5.471,149.139
C00514=1207.644,-92.113,-38.508,179.398,5.471,149.139
C00515=1207.649,-92.363,-38.497,179.395,5.471,149.140
C00516=1207.655,-92.613,-38.487,179.393,5.471,149.141
C00517=1207.660,-92.863,-38.476,179.390,5.471,149.142
C00518=1207.666,-93.112,-38.466,179.388,5.471,149.142
C00519=1207.670,-93.362,-38.455,179.386,5.470,149.143
C00520=1207.676,-93.612,-38.444,179.384,5.471,149.143
C00521=1207.682,-93.861,-38.434,179.381,5.470,149.144
C00522=1207.687,-94.111,-38.424,179.378,5.470,149.145
C00523=1207.692,-94.361,-38.413,179.377,5.470,149.145
C00524=1207.696,-94.611,-38.403,179.374,5.470,149.146
C00525=1207.702,-94.860,-38.393,179.372,5.470,149.147
C00526=1207.708,-95.110,-38.383,179.369,5.470,149.147
C00527=1207.713,-95.360,-38.372,179.367,5.470,149.148
C00528=1207.718,-95.609,-38.362,179.365,5.469,149.149
C00529=1207.723,-95.859,-38.351,179.363,5.469,149.149
C00530=1207.728,-96.109,-38.341,179.360,5.469,149.150
C00531=1207.734,-96.358,-38.331,179.358,5.469,149.151
C00532=1207.738,-96.608,-38.321,179.356,5.469,149.152
C00533=1207.744,-96.858,-38.310,179.354,5.469,149.152
C00534=1207.749,-97.108,-38.300,179.351,5.469,149.153
C00535=1207.755,-97.358,-38.290,179.349,5.469,149.153
C00536=1207.760,-97.607,-38.279,179.347,5.469,149.154
C00537=1207.765,-97.857,-38.269,179.345,5.469,149.155
C00538=1207.771,-98.107,-38.259,179.342,5.468,149.155
C00539=1207.776,-98.356,-38.249,179.340,5.468,149.156
C00540=1207.781,-98.606,-38.238,179.338,5.468,149.157
C00541=1207.786,-98.856,-38.228,179.335,5.468,149.157
C00542=1207.792,-99.106,-38.218,179.333,5.468,149.158
C00543=1207.797,-99.356,-38.207,179.331,5.468,149.159
C00544=1207.802,-99.605,-38.198,179.329,5.468,149.159
C00545=1207.807,-99.855,-38.188,179.326,5.468,149.160
C00546=1207.812,-100.105,-38.177,179.324,5.467,149.161
C00547=1207.818,-100.354,-38.167,179.322,5.468,149.161
C00548=1207.823,-100.604,-38.157,179.319,5.467,149.162
C00549=1207.829,-100.875,-38.146,179.317,5.467,149.163
C00550=1207.834,-101.147,-38.135,179.315,5.467,149.163
C00551=1207.840,-101.418,-38.123,179.312,5.467,149.164
C00552=1207.846,-101.689,-38.113,179.309,5.466,149.165
C00553=1207.851,-101.940,-38.103,179.307,5.467,149.166
C00554=1207.856,-102.189,-38.093,179.305,5.466,149.166
C00555=1207.861,-102.438,-38.083,179.303,5.466,149.167
C00556=1207.866,-102.689,-38.072,179.300,5.466,149.167
C00557=1207.872,-102.938,-38.062,179.298,5.466,149.168
C00558=1207.877,-103.188,-38.052,179.296,5.465,149.169
C00559=1207.882,-103.438,-38.042,179.294,5.466,149.169
C00560=1207.887,-103.687,-38.032,179.291,5.465,149.170
C00561=1207.893,-103.937,-38.022,179.289,5.466,149.171
C00562=1207.898,-104.187,-38.013,179.287,5.465,149.171
C00563=1207.903,-104.437,-38.002,179.285,5.465,149.172
C00564=1207.909,-104.686,-37.992,179.282,5.465,149.173
C00565=1207.914,-104.936,-37.982,179.280,5.465,149.173
C00566=1207.919,-105.186,-37.972,179.278,5.464,149.174
C00567=1207.924,-105.436,-37.962,179.276,5.465,149.175
C00568=1207.930,-105.686,-37.952,179.273,5.464,149.175
C00569=1207.935,-105.935,-37.942,179.271,5.465,149.176
C00570=1207.940,-106.185,-37.932,179.269,5.464,149.177
C00571=1207.945,-106.435,-37.922,179.267,5.464,149.177
C00572=1207.951,-106.684,-37.913,179.264,5.464,149.178
C00573=1207.956,-106.934,-37.902,179.262,5.464,149.179
C00574=1207.961,-107.184,-37.892,179.260,5.464,149.179
C00575=1207.966,-107.433,-37.882,179.258,5.464,149.180
C00576=1207.972,-107.683,-37.872,179.255,5.464,149.181
C00577=1207.978,-107.933,-37.863,179.253,5.464,149.181
C00578=1207.982,-108.183,-37.853,179.251,5.463,149.182
C00579=1207.987,-108.433,-37.842,179.249,5.464,149.183
C00580=1207.993,-108.682,-37.834,179.246,5.463,149.183
C00581=1207.998,-108.932,-37.823,179.244,5.464,149.184
C00582=1208.004,-109.182,-37.813,179.242,5.464,149.184
C00583=1208.008,-109.431,-37.803,179.240,5.463,149.185
C00584=1208.014,-109.682,-37.794,179.238,5.464,149.186
C00585=1208.019,-109.931,-37.784,179.235,5.463,149.187
C00586=1208.024,-110.180,-37.774,179.233,5.463,149.187
C00587=1208.030,-110.431,-37.764,179.231,5.463,149.188
C00588=1208.035,-110.681,-37.754,179.229,5.463,149.188
C00589=1208.040,-110.930,-37.744,179.226,5.463,149.189
C00590=1208.045,-111.180,-37.735,179.224,5.463,149.190
C00591=1208.051,-111.429,-37.725,179.222,5.462,149.190
C00592=1208.057,-111.679,-37.715,179.220,5.463,149.191
C00593=1208.061,-111.930,-37.706,179.217,5.462,149.192
C00594=1208.067,-112.179,-37.695,179.215,5.462,149.192
C00595=1208.072,-112.428,-37.686,179.213,5.462,149.193
C00596=1208.078,-112.678,-37.676,179.210,5.462,149.194
C00597=1208.082,-112.928,-37.667,179.208,5.461,149.194
C00598=1208.088,-113.177,-37.656,179.206,5.462,149.195
C00599=1208.093,-113.428,-37.647,179.204,5.461,149.196
C00600=1208.098,-113.677,-37.637,179.202,5.461,149.196
C00601=1208.103,-113.927,-37.628,179.199,5.461,149.197
C00602=1208.109,-114.177,-37.618,179.197,5.461,149.198
C00603=1208.114,-114.426,-37.608,179.194,5.461,149.198
C00604=1208.120,-114.676,-37.599,179.193,5.461,149.199
C00605=1208.125,-114.925,-37.589,179.190,5.461,149.199
C00606=1208.130,-115.176,-37.579,179.188,5.461,149.200
C00607=1208.135,-115.425,-37.570,179.186,5.460,149.201
C00608=1208.141,-115.676,-37.560,179.184,5.461,149.201
C00609=1208.145,-115.925,-37.551,179.181,5.460,149.202
C00610=1208.151,-116.175,-37.541,179.179,5.461,149.203
C00611=1208.156,-116.424,-37.531,179.177,5.460,149.203
C00612=1208.162,-116.674,-37.522,179.175,5.460,149.204
C00613=1208.166,-116.924,-37.512,179.173,5.461,149.205
C00614=1208.172,-117.175,-37.502,179.170,5.460,149.205
C00615=1208.177,-117.424,-37.493,179.168,5.460,149.206
C00616=1208.183,-117.674,-37.483,179.166,5.460,149.207
C00617=1208.188,-117.923,-37.474,179.164,5.460,149.207
C00618=1208.194,-118.173,-37.464,179.161,5.459,149.208
C00619=1208.199,-118.423,-37.455,179.159,5.460,149.209
C00620=1208.204,-118.672,-37.446,179.157,5.459,149.209
C00621=1208.209,-118.922,-37.436,179.155,5.459,149.210
C00622=1208.215,-119.172,-37.427,179.152,5.459,149.211
C00623=1208.220,-119.422,-37.416,179.150,5.459,149.211
C00624=1208.225,-119.672,-37.407,179.148,5.458,149.212
C00625=1208.230,-119.921,-37.397,179.146,5.459,149.212
C00626=1208.236,-120.171,-37.388,179.143,5.458,149.213
C00627=1208.240,-120.420,-37.378,179.142,5.458,149.214
C00628=1208.246,-120.671,-37.369,179.139,5.458,149.214
C00629=1208.251,-120.921,-37.360,179.137,5.458,149.215
C00630=1208.256,-121.170,-37.350,179.135,5.459,149.216
C00631=1208.262,-121.420,-37.341,179.133,5.458,149.216
C00632=1208.267,-121.669,-37.331,179.131,5.458,149.217
C00633=1208.273,-121.919,-37.322,179.128,5.458,149.218
C00634=1208.278,-122.169,-37.313,179.126,5.458,149.218
C00635=1208.283,-122.418,-37.303,179.124,5.458,149.219
C00636=1208.289,-122.669,-37.294,179.122,5.458,149.220
C00637=1208.294,-122.918,-37.285,179.119,5.457,149.220
C00638=1208.299,-123.168,-37.275,179.117,5.458,149.221
C00639=1208.304,-123.419,-37.265,179.115,5.457,149.222
C00640=1208.309,-123.668,-37.257,179.113,5.457,149.222
C00641=1208.314,-123.918,-37.247,179.110,5.457,149.223
C00642=1208.320,-124.168,-37.237,179.108,5.457,149.223
C00643=1208.325,-124.418,-37.229,179.107,5.457,149.224
C00644=1208.330,-124.667,-37.219,179.104,5.457,149.225
C00645=1208.336,-124.917,-37.209,179.102,5.457,149.225
C00646=1208.341,-125.167,-37.201,179.100,5.456,149.226
C00647=1208.346,-125.416,-37.191,179.098,5.457,149.227
C00648=1208.352,-125.666,-37.181,179.095,5.456,149.227
C00649=1208.357,-125.916,-37.173,179.093,5.456,149.228
C00650=1208.362,-126.166,-37.164,179.091,5.456,149.228
C00651=1208.367,-126.415,-37.154,179.089,5.456,149.229
C00652=1208.373,-126.665,-37.145,179.086,5.456,149.230
C00653=1207.952,-126.676,-37.183,179.082,5.459,149.232
C00654=1207.946,-126.426,-37.191,179.085,5.460,149.231
C00655=1207.942,-126.177,-37.201,179.087,5.459,149.230
C00656=1207.936,-125.926,-37.211,179.089,5.460,149.230
C00657=1207.930,-125.677,-37.219,179.091,5.460,149.229
C00658=1207.925,-125.427,-37.228,179.094,5.460,149.228
C00659=1207.920,-125.177,-37.239,179.095,5.460,149.228
C00660=1207.915,-124.927,-37.247,179.098,5.460,149.227
C00661=1207.909,-124.677,-37.256,179.100,5.460,149.227
C00662=1207.905,-124.428,-37.266,179.102,5.461,149.226
C00663=1207.899,-124.178,-37.275,179.104,5.460,149.225
C00664=1207.893,-123.928,-37.284,179.106,5.460,149.225
C00665=1207.889,-123.679,-37.294,179.109,5.461,149.224
C00666=1207.883,-123.429,-37.303,179.111,5.460,149.223
C00667=1207.878,-123.179,-37.312,179.113,5.461,149.223
C00668=1207.873,-122.930,-37.322,179.115,5.461,149.222
C00669=1207.867,-122.680,-37.331,179.118,5.461,149.221
C00670=1207.862,-122.430,-37.340,179.120,5.461,149.221
C00671=1207.856,-122.180,-37.351,179.122,5.462,149.220
C00672=1207.851,-121.930,-37.359,179.124,5.461,149.220
C00673=1207.846,-121.681,-37.368,179.127,5.462,149.219
C00674=1207.840,-121.431,-37.379,179.128,5.462,149.218
C00675=1207.835,-121.181,-37.387,179.131,5.462,149.218
C00676=1207.831,-120.931,-37.397,179.133,5.462,149.217
C00677=1207.825,-120.681,-37.407,179.135,5.462,149.216
C00678=1207.820,-120.431,-37.416,179.137,5.462,149.216
C00679=1207.814,-120.182,-37.426,179.139,5.462,149.215
C00680=1207.809,-119.932,-37.435,179.142,5.462,149.215
C00681=1207.804,-119.683,-37.445,179.144,5.462,149.214
C00682=1207.798,-119.432,-37.454,179.146,5.462,149.213
C00683=1207.793,-119.183,-37.464,179.148,5.462,149.212
C00684=1207.787,-118.933,-37.473,179.151,5.463,149.212
C00685=1207.782,-118.683,-37.482,179.153,5.462,149.211
C00686=1207.777,-118.434,-37.492,179.155,5.463,149.210
C00687=1207.771,-118.184,-37.501,179.157,5.463,149.210
C00688=1207.767,-117.934,-37.511,179.160,5.463,149.209
C00689=1207.761,-117.684,-37.521,179.162,5.463,149.209
C00690=1207.756,-117.434,-37.530,179.164,5.464,149.208
C00691=1207.750,-117.184,-37.540,179.166,5.463,149.207
C00692=1207.746,-116.935,-37.549,179.169,5.464,149.207
C00693=1207.740,-116.685,-37.558,179.170,5.464,149.206
C00694=1207.735,-116.436,-37.568,179.173,5.464,149.205
C00695=1207.730,-116.186,-37.577,179.175,5.464,149.205
C00696=1207.724,-115.936,-37.588,179.177,5.463,149.204
C00697=1207.719,-115.686,-37.597,179.179,5.464,149.203
C00698=1207.714,-115.436,-37.607,179.181,5.464,149.203
C00699=1207.709,-115.187,-37.617,179.184,5.464,149.202
C00700=1207.703,-114.937,-37.626,179.186,5.464,149.202
C00701=1207.698,-114.688,-37.636,179.188,5.465,149.201
C00702=1207.692,-114.437,-37.645,179.191,5.464,149.200
C00703=1207.687,-114.188,-37.655,179.193,5.465,149.199
C00704=1207.682,-113.937,-37.665,179.195,5.465,149.199
C00705=1207.677,-113.688,-37.674,179.197,5.465,149.198
C00706=1207.672,-113.438,-37.685,179.200,5.465,149.198
C00707=1207.666,-113.188,-37.694,179.202,5.465,149.197
C00708=1207.661,-112.939,-37.704,179.204,5.465,149.196
C00709=1207.655,-112.689,-37.713,179.207,5.465,149.196
C00710=1207.650,-112.440,-37.723,179.209,5.465,149.195
C00711=1207.645,-112.189,-37.733,179.211,5.466,149.194
C00712=1207.640,-111.940,-37.742,179.213,5.465,149.194
C00713=1207.634,-111.690,-37.752,179.216,5.466,149.193
C00714=1207.630,-111.441,-37.762,179.217,5.466,149.192
C00715=1207.624,-111.191,-37.772,179.220,5.466,149.192
C00716=1207.619,-110.941,-37.782,179.222,5.466,149.191
C00717=1207.614,-110.691,-37.792,179.225,5.466,149.190
C00718=1207.608,-110.441,-37.801,179.226,5.466,149.190
C00719=1207.603,-110.192,-37.811,179.229,5.467,149.189
C00720=1207.597,-109.942,-37.821,179.231,5.466,149.188
C00721=1207.593,-109.692,-37.830,179.234,5.467,149.188
C00722=1207.587,-109.442,-37.841,179.235,5.467,149.187
C00723=1207.582,-109.193,-37.851,179.238,5.467,149.187
C00724=1207.576,-108.943,-37.860,179.240,5.467,149.186
C00725=1207.571,-108.693,-37.870,179.242,5.467,149.185
C00726=1207.567,-108.443,-37.880,179.244,5.467,149.185
C00727=1207.561,-108.194,-37.890,179.247,5.468,149.184
C00728=1207.555,-107.944,-37.900,179.249,5.467,149.183
C00729=1207.550,-107.694,-37.909,179.251,5.468,149.183
C00730=1207.545,-107.444,-37.920,179.253,5.468,149.182
C00731=1207.540,-107.195,-37.930,179.256,5.468,149.181
C00732=1207.535,-106.945,-37.939,179.258,5.468,149.181
C00733=1207.529,-106.695,-37.949,179.260,5.468,149.180
C00734=1207.524,-106.445,-37.960,179.262,5.468,149.179
C00735=1207.519,-106.196,-37.969,179.264,5.468,149.179
C00736=1207.513,-105.946,-37.979,179.267,5.468,149.178
C00737=1207.508,-105.696,-37.989,179.269,5.468,149.177
C00738=1207.503,-105.446,-37.999,179.271,5.468,149.177
C00739=1207.498,-105.196,-38.009,179.274,5.468,149.176
C00740=1207.492,-104.947,-38.019,179.276,5.468,149.175
C00741=1207.487,-104.698,-38.029,179.278,5.468,149.175
C00742=1207.482,-104.447,-38.039,179.280,5.469,149.174
C00743=1207.476,-104.197,-38.049,179.283,5.468,149.173
C00744=1207.471,-103.948,-38.059,179.285,5.469,149.173
C00745=1207.466,-103.699,-38.069,179.287,5.469,149.172
C00746=1207.461,-103.448,-38.079,179.290,5.469,149.171
C00747=1207.455,-103.199,-38.090,179.292,5.470,149.171
C00748=1207.450,-102.950,-38.099,179.294,5.469,149.170
C00749=1207.445,-102.699,-38.109,179.296,5.470,149.170
C00750=1207.440,-102.449,-38.119,179.299,5.470,149.169
C00751=1207.435,-102.200,-38.129,179.301,5.470,149.168
C00752=1207.430,-101.950,-38.139,179.303,5.470,149.167
C00753=1207.424,-101.700,-38.150,179.306,5.471,149.167
C00754=1207.419,-101.429,-38.161,179.308,5.470,149.166
C00755=1207.412,-101.158,-38.172,179.310,5.471,149.166
C00756=1207.407,-100.887,-38.183,179.312,5.470,149.165
C00757=1207.401,-100.615,-38.194,179.315,5.471,149.164
C00758=1207.396,-100.366,-38.204,179.318,5.471,149.163
C00759=1207.390,-100.116,-38.213,179.320,5.471,149.163
C00760=1207.385,-99.865,-38.224,179.322,5.471,149.162
C00761=1207.380,-99.616,-38.234,179.324,5.471,149.161
C00762=1207.375,-99.367,-38.244,179.327,5.472,149.161
C00763=1207.370,-99.116,-38.254,179.329,5.471,149.160
C00764=1207.364,-98.867,-38.265,179.332,5.472,149.159
C00765=1207.359,-98.617,-38.275,179.334,5.471,149.159
C00766=1207.354,-98.367,-38.285,179.336,5.472,149.158
C00767=1207.348,-98.117,-38.296,179.338,5.472,149.157
C00768=1207.344,-97.867,-38.306,179.341,5.472,149.157
C00769=1207.338,-97.618,-38.316,179.343,5.472,149.156
C00770=1207.333,-97.368,-38.326,179.345,5.472,149.156
C00771=1207.328,-97.118,-38.337,179.347,5.472,149.155
C00772=1207.322,-96.869,-38.347,179.350,5.473,149.154
C00773=1207.317,-96.619,-38.357,179.352,5.472,149.153
C00774=1207.313,-96.370,-38.368,179.354,5.473,149.153
C00775=1207.307,-96.120,-38.378,179.356,5.473,149.152
C00776=1207.302,-95.870,-38.388,179.359,5.473,149.151
C00777=1207.296,-95.620,-38.399,179.361,5.473,149.151
C00778=1207.291,-95.371,-38.409,179.363,5.473,149.150
C00779=1207.286,-95.121,-38.419,179.365,5.473,149.150
C00780=1207.280,-94.871,-38.430,179.368,5.473,149.149
C00781=1207.275,-94.621,-38.440,179.370,5.474,149.148
C00782=1207.270,-94.372,-38.450,179.372,5.473,149.147
C00783=1207.265,-94.122,-38.460,179.375,5.474,149.147
C00784=1207.260,-93.872,-38.471,179.377,5.474,149.146
C00785=1207.254,-93.623,-38.482,179.379,5.474,149.146
C00786=1207.249,-93.373,-38.492,179.381,5.474,149.145
C00787=1207.244,-93.123,-38.502,179.384,5.474,149.144
C00788=1207.238,-92.874,-38.513,179.386,5.474,149.144
C00789=1207.233,-92.623,-38.523,179.388,5.475,149.143
C00790=1207.228,-92.374,-38.533,179.391,5.474,149.142
C00791=1207.223,-92.124,-38.544,179.393,5.475,149.141
C00792=1207.217,-91.875,-38.555,179.395,5.474,149.141
C00793=1207.212,-91.624,-38.565,179.397,5.475,149.140
C00794=1207.207,-91.375,-38.576,179.400,5.475,149.140
C00795=1207.201,-91.125,-38.586,179.402,5.475,149.139
C00796=1207.197,-90.875,-38.596,179.404,5.475,149.138
C00797=1207.192,-90.626,-38.607,179.407,5.475,149.137
C00798=1207.187,-90.376,-38.617,179.409,5.476,149.137
C00799=1207.181,-90.127,-38.627,179.411,5.476,149.136
C00800=1207.176,-89.876,-38.638,179.414,5.476,149.136
C00801=1207.170,-89.627,-38.648,179.416,5.476,149.135
C00802=1207.166,-89.377,-38.660,179.418,5.477,149.134
C00803=1207.160,-89.128,-38.670,179.420,5.476,149.134
C00804=1207.155,-88.877,-38.680,179.423,5.477,149.133
C00805=1207.150,-88.628,-38.691,179.425,5.476,149.132
C00806=1207.145,-88.378,-38.702,179.428,5.477,149.131
C00807=1207.139,-88.129,-38.712,179.429,5.477,149.131
C00808=1207.134,-87.878,-38.723,179.432,5.477,149.130
C00809=1207.129,-87.630,-38.734,179.434,5.477,149.130
C00810=1207.124,-87.379,-38.744,179.437,5.477,149.129
C00811=1207.118,-87.130,-38.754,179.439,5.478,149.128
C00812=1207.114,-86.880,-38.766,179.441,5.478,149.128
C00813=1207.107,-86.630,-38.776,179.444,5.478,149.127
C00814=1207.102,-86.380,-38.787,179.446,5.478,149.126
C00815=1207.097,-86.131,-38.798,179.448,5.478,149.126
C00816=1207.092,-85.881,-38.808,179.451,5.478,149.125
C00817=1207.086,-85.631,-38.819,179.453,5.478,149.124
C00818=1207.082,-85.382,-38.830,179.455,5.478,149.124
C00819=1207.076,-85.132,-38.840,179.457,5.479,149.123
C00820=1207.071,-84.882,-38.851,179.460,5.478,149.122
C00821=1207.066,-84.633,-38.862,179.462,5.479,149.122
C00822=1207.061,-84.383,-38.872,179.465,5.479,149.121
C00823=1207.056,-84.133,-38.883,179.467,5.479,149.120
C00824=1207.051,-83.884,-38.894,179.469,5.480,149.120
C00825=1207.046,-83.633,-38.904,179.471,5.479,149.119
C00826=1207.040,-83.384,-38.915,179.474,5.480,149.118
C00827=1207.035,-83.134,-38.926,179.476,5.479,149.117
C00828=1207.029,-82.884,-38.937,179.478,5.480,149.117
C00829=1207.024,-82.635,-38.948,179.480,5.480,149.116
C00830=1207.019,-82.385,-38.958,179.483,5.480,149.116
C00831=1207.014,-82.136,-38.969,179.486,5.481,149.115
C00832=1207.009,-81.885,-38.980,179.488,5.480,149.114
C00833=1207.004,-81.636,-38.991,179.490,5.481,149.113
C00834=1206.998,-81.386,-39.002,179.492,5.481,149.113
C00835=1206.993,-81.137,-39.013,179.495,5.481,149.112
C00836=1206.988,-80.887,-39.024,179.497,5.481,149.112
C00837=1206.982,-80.638,-39.035,179.499,5.481,149.111
C00838=1206.977,-80.387,-39.045,179.502,5.481,149.110
C00839=1206.973,-80.138,-39.056,179.504,5.482,149.110
C00840=1206.966,-79.888,-39.067,179.506,5.482,149.109
C00841=1206.962,-79.638,-39.078,179.508,5.482,149.108
C00842=1206.956,-79.389,-39.089,179.511,5.482,149.108
C00843=1206.951,-79.139,-39.100,179.513,5.482,149.107
C00844=1206.946,-78.889,-39.111,179.516,5.482,149.106
C00845=1206.941,-78.640,-39.121,179.517,5.482,149.106
C00846=1206.935,-78.389,-39.133,179.520,5.483,149.105
C00847=1206.931,-78.140,-39.144,179.523,5.483,149.104
C00848=1206.925,-77.890,-39.154,179.525,5.483,149.104
C00849=1206.920,-77.641,-39.165,179.528,5.483,149.103
C00850=1206.914,-77.391,-39.176,179.529,5.483,149.102
C00851=1206.909,-77.141,-39.188,179.532,5.484,149.102
C00852=1206.905,-76.892,-39.199,179.534,5.483,149.101
C00853=1206.899,-76.642,-39.209,179.537,5.484,149.100
C00854=1206.894,-76.392,-39.221,179.539,5.484,149.099
C00855=1206.889,-76.142,-39.232,179.541,5.484,149.099
C00856=1206.883,-75.893,-39.242,179.544,5.485,149.098
C00857=1206.879,-75.643,-39.254,179.546,5.484,149.098
C00858=1206.873,-75.372,-39.266,179.548,5.485,149.097
C00859=1206.867,-75.102,-39.278,179.551,5.485,149.096
C00860=1206.861,-74.831,-39.290,179.553,5.485,149.095
C00861=1206.855,-74.561,-39.302,179.556,5.485,149.095
C00862=1206.850,-74.311,-39.313,179.558,5.486,149.094
C00863=1206.845,-74.061,-39.324,179.560,5.485,149.093
C00864=1206.841,-73.811,-39.335,179.563,5.486,149.093
C00865=1206.834,-73.561,-39.346,179.565,5.485,149.092
C00866=1206.830,-73.312,-39.357,179.568,5.486,149.091
C00867=1206.825,-73.062,-39.369,179.571,5.486,149.091
C00868=1206.819,-72.813,-39.380,179.572,5.486,149.090
C00869=1206.814,-72.563,-39.391,179.575,5.487,149.089
C00870=1206.809,-72.313,-39.402,179.577,5.486,149.089
C00871=1206.803,-72.064,-39.413,179.580,5.487,149.088
C00872=1206.798,-71.814,-39.424,179.582,5.486,149.087
C00873=1206.793,-71.564,-39.435,179.584,5.487,149.086
C00874=1206.787,-71.315,-39.447,179.587,5.488,149.086
C00875=1206.783,-71.065,-39.458,179.589,5.487,149.085
C00876=1206.777,-70.815,-39.469,179.591,5.488,149.085
C00877=1206.772,-70.565,-39.481,179.593,5.487,149.084
C00878=1206.767,-70.316,-39.491,179.596,5.488,149.083
C00879=1206.762,-70.066,-39.503,179.599,5.488,149.082
C00880=1206.757,-69.816,-39.515,179.600,5.488,149.082
C00881=1206.752,-69.566,-39.525,179.603,5.489,149.081
C00882=1206.746,-69.317,-39.537,179.605,5.488,149.081
C00883=1206.741,-69.067,-39.548,179.608,5.489,149.080
C00884=1206.736,-68.817,-39.560,179.610,5.489,149.079
C00885=1206.731,-68.568,-39.571,179.613,5.489,149.078
C00886=1206.725,-68.318,-39.582,179.615,5.489,149.078
C00887=1206.720,-68.068,-39.593,179.617,5.489,149.077
C00888=1206.715,-67.819,-39.605,179.619,5.490,149.077
C00889=1206.710,-67.569,-39.616,179.622,5.490,149.076
C00890=1206.705,-67.320,-39.627,179.624,5.490,149.075
C00891=1206.699,-67.070,-39.639,179.627,5.490,149.074
C00892=1206.694,-66.820,-39.651,179.629,5.490,149.074
C00893=1206.689,-66.570,-39.662,179.631,5.491,149.073
C00894=1206.683,-66.321,-39.673,179.634,5.491,149.073
C00895=1206.679,-66.071,-39.684,179.636,5.491,149.072
C00896=1206.673,-65.821,-39.696,179.639,5.491,149.071
C00897=1206.669,-65.572,-39.707,179.641,5.491,149.070
C00898=1206.663,-65.322,-39.719,179.643,5.491,149.070
C00899=1206.658,-65.073,-39.730,179.646,5.492,149.069
C00900=1206.652,-64.823,-39.742,179.648,5.492,149.069
C00901=1206.648,-64.573,-39.753,179.650,5.492,149.068
C00902=1206.642,-64.323,-39.765,179.652,5.492,149.067
C00903=1206.638,-64.074,-39.776,179.655,5.492,149.066
C00904=1206.632,-63.824,-39.788,179.658,5.493,149.066
C00905=1206.627,-63.575,-39.799,179.660,5.492,149.065
C00906=1206.621,-63.324,-39.810,179.662,5.493,149.064
C00907=1206.617,-63.075,-39.822,179.664,5.493,149.064
C00908=1206.611,-62.825,-39.833,179.667,5.493,149.063
C00909=1206.606,-62.575,-39.845,179.669,5.494,149.062
C00910=1206.600,-62.326,-39.856,179.671,5.493,149.062
C00911=1206.595,-62.076,-39.868,179.674,5.494,149.061
C00912=1206.590,-61.826,-39.879,179.677,5.494,149.060
C00913=1206.585,-61.576,-39.891,179.679,5.494,149.060
C00914=1206.580,-61.327,-39.903,179.681,5.495,149.059
C00915=1206.575,-61.077,-39.915,179.683,5.494,149.058
C00916=1206.570,-60.828,-39.927,179.686,5.495,149.058
C00917=1206.564,-60.578,-39.938,179.688,5.495,149.057
C00918=1206.560,-60.329,-39.949,179.691,5.495,149.056
C00919=1206.554,-60.079,-39.961,179.693,5.495,149.056
C00920=1206.549,-59.829,-39.973,179.695,5.495,149.055
C00921=1206.544,-59.579,-39.984,179.697,5.496,149.054
C00922=1206.539,-59.329,-39.996,179.700,5.496,149.054
C00923=1206.534,-59.080,-40.008,179.702,5.496,149.053
C00924=1206.528,-58.830,-40.019,179.705,5.496,149.052
C00925=1206.522,-58.581,-40.031,179.708,5.497,149.052
C00926=1206.518,-58.331,-40.042,179.710,5.497,149.051
C00927=1206.513,-58.082,-40.055,179.712,5.497,149.050
C00928=1206.508,-57.832,-40.066,179.714,5.497,149.050
C00929=1206.503,-57.582,-40.078,179.717,5.498,149.049
C00930=1206.497,-57.332,-40.090,179.719,5.498,149.048
C00931=1206.492,-57.083,-40.101,179.721,5.498,149.048
C00932=1206.487,-56.833,-40.113,179.724,5.498,149.047
C00933=1206.482,-56.583,-40.125,179.727,5.499,149.046
C00934=1206.477,-56.334,-40.137,179.729,5.498,149.045
C00935=1206.472,-56.084,-40.149,179.731,5.499,149.045
C00936=1206.466,-55.834,-40.161,179.734,5.499,149.044
C00937=1206.462,-55.584,-40.172,179.736,5.499,149.044
C00938=1206.456,-55.335,-40.184,179.738,5.500,149.043
C00939=1206.450,-55.086,-40.196,179.740,5.499,149.042
C00940=1206.446,-54.836,-40.207,179.743,5.500,149.041
C00941=1206.440,-54.586,-40.219,179.746,5.500,149.041
C00942=1206.435,-54.336,-40.231,179.747,5.500,149.040
C00943=1206.431,-54.087,-40.243,179.750,5.501,149.040
C00944=1206.425,-53.837,-40.255,179.753,5.501,149.039
C00945=1206.420,-53.587,-40.267,179.755,5.501,149.038
C00946=1206.415,-53.338,-40.278,179.757,5.501,149.037
C00947=1206.410,-53.088,-40.291,179.760,5.502,149.037
C00948=1206.404,-52.838,-40.303,179.762,5.501,149.036
C00949=1206.399,-52.588,-40.315,179.765,5.502,149.035
C00950=1206.394,-52.339,-40.326,179.766,5.502,149.035
C00951=1206.389,-52.089,-40.339,179.769,5.502,149.034
C00952=1206.384,-51.840,-40.350,179.772,5.503,149.034
C00953=1206.378,-51.590,-40.362,179.774,5.502,149.033
C00954=1206.374,-51.341,-40.374,179.777,5.503,149.032
C00955=1206.368,-51.091,-40.386,179.779,5.503,149.031
C00956=1206.363,-50.841,-40.398,179.781,5.503,149.031
C00957=1206.358,-50.591,-40.411,179.783,5.504,149.030
C00958=1206.353,-50.342,-40.422,179.786,5.504,149.030
C00959=1206.348,-50.092,-40.434,179.788,5.504,149.029
C00960=1206.343,-49.843,-40.446,179.791,5.504,149.028
C00961=1206.337,-49.593,-40.458,179.794,5.505,149.027
C00962=1206.332,-49.322,-40.471,179.796,5.504,149.027
C00963=1206.326,-49.053,-40.484,179.798,5.505,149.026
C00964=1206.321,-48.783,-40.498,179.801,5.505,149.025
C00965=1206.316,-48.512,-40.511,179.804,5.506,149.025
C00966=1206.310,-48.263,-40.522,179.806,5.505,149.024
C00967=1206.305,-48.013,-40.535,179.808,5.506,149.023
C00968=1206.300,-47.763,-40.547,179.811,5.506,149.022
C00969=1206.295,-47.514,-40.560,179.813,5.506,149.022
C00970=1206.289,-47.264,-40.571,179.816,5.506,149.021
C00971=1206.284,-47.014,-40.583,179.818,5.507,149.020
C00972=1206.279,-46.765,-40.595,179.820,5.507,149.020
C00973=1206.274,-46.515,-40.607,179.823,5.507,149.019
C00974=1206.269,-46.266,-40.620,179.825,5.508,149.019
C00975=1206.263,-46.016,-40.632,179.827,5.507,149.018
C00976=1206.258,-45.767,-40.644,179.830,5.508,149.017
C00977=1206.253,-45.517,-40.656,179.833,5.508,149.016
C00978=1206.248,-45.267,-40.669,179.835,5.508,149.016
C00979=1206.242,-45.017,-40.681,179.838,5.509,149.015
C00980=1206.238,-44.768,-40.693,179.840,5.509,149.015
C00981=1206.232,-44.518,-40.705,179.842,5.509,149.014
C00982=1206.228,-44.268,-40.718,179.844,5.509,149.013
C00983=1206.223,-44.018,-40.729,179.847,5.510,149.012
C00984=1206.217,-43.769,-40.742,179.850,5.510,149.012
C00985=1206.212,-43.519,-40.754,179.852,5.510,149.011
C00986=1206.207,-43.270,-40.766,179.855,5.511,149.010
C00987=1206.202,-43.021,-40.779,179.857,5.511,149.010
C00988=1206.196,-42.771,-40.791,179.859,5.511,149.009
C00989=1206.191,-42.521,-40.804,179.861,5.511,149.008
C00990=1206.186,-42.271,-40.815,179.864,5.512,149.008
C00991=1206.181,-42.021,-40.828,179.866,5.512,149.007
C00992=1206.176,-41.771,-40.840,179.869,5.512,149.006
C00993=1206.171,-41.522,-40.853,179.872,5.513,149.006
C00994=1206.166,-41.273,-40.866,179.874,5.512,149.005
C00995=1206.160,-41.023,-40.877,179.876,5.513,149.004
C00996=1206.155,-40.774,-40.890,179.878,5.513,149.004
C00997=1206.150,-40.524,-40.903,179.881,5.513,149.003
C00998=1206.145,-40.274,-40.915,179.883,5.514,149.002
C00999=1206.140,-40.024,-40.927,179.886,5.514,149.002
C01000=1206.135,-39.775,-40.940,179.888,5.514,149.001
C01001=1206.129,-39.525,-40.952,179.891,5.514,149.000
C01002=1206.124,-39.276,-40.965,179.893,5.515,149.000
C01003=1206.119,-39.026,-40.977,179.896,5.515,148.999
C01004=1206.114,-38.776,-40.989,179.897,5.515,148.998
C01005=1206.109,-38.526,-41.002,179.900,5.516,148.998
C01006=1206.104,-38.277,-41.015,179.903,5.516,148.997
C01007=1206.099,-38.027,-41.026,179.905,5.516,148.996
C01008=1206.093,-37.778,-41.039,179.908,5.516,148.996
C01009=1206.088,-37.529,-41.052,179.910,5.517,148.995
C01010=1206.084,-37.279,-41.065,179.912,5.516,148.994
C01011=1206.078,-37.029,-41.077,179.915,5.517,148.993
C01012=1206.073,-36.779,-41.089,179.918,5.517,148.993
C01013=1206.068,-36.530,-41.102,179.920,5.518,148.992
C01014=1206.063,-36.281,-41.114,179.922,5.518,148.992
C01015=1206.058,-36.031,-41.126,179.925,5.518,148.991
C01016=1206.052,-35.780,-41.140,179.927,5.519,148.990
C01017=1206.047,-35.531,-41.152,179.929,5.518,148.990
C01018=1206.042,-35.282,-41.165,179.932,5.519,148.989
C01019=1206.037,-35.032,-41.177,179.935,5.519,148.988
C01020=1206.032,-34.782,-41.190,179.937,5.519,148.987
C01021=1206.027,-34.532,-41.202,179.939,5.520,148.987
C01022=1206.022,-34.283,-41.215,179.942,5.520,148.986
C01023=1206.017,-34.034,-41.228,179.944,5.521,148.986
C01024=1206.011,-33.784,-41.241,179.946,5.520,148.985
C01025=1206.006,-33.534,-41.253,179.949,5.521,148.984
C01026=1206.001,-33.284,-41.266,179.952,5.521,148.983
C01027=1205.996,-33.035,-41.278,179.954,5.521,148.983
C01028=1205.991,-32.786,-41.291,179.956,5.522,148.982
C01029=1205.986,-32.536,-41.304,179.959,5.522,148.982
C01030=1205.981,-32.286,-41.316,179.961,5.523,148.981
C01031=1205.975,-32.037,-41.330,179.963,5.523,148.980
C01032=1205.970,-31.787,-41.342,179.966,5.523,148.980
C01033=1205.965,-31.537,-41.355,179.969,5.523,148.979
C01034=1205.960,-31.287,-41.367,179.971,5.523,148.978
C01035=1205.955,-31.038,-41.380,179.973,5.524,148.977
C01036=1205.950,-30.788,-41.393,179.976,5.524,148.977
C01037=1205.945,-30.538,-41.406,179.978,5.525,148.976
C01038=1205.939,-30.289,-41.418,179.980,5.525,148.976
C01039=1205.934,-30.040,-41.431,179.983,5.525,148.975
C01040=1205.930,-29.790,-41.444,179.986,5.526,148.974
C01041=1205.924,-29.540,-41.457,179.988,5.526,148.973
C01042=1205.919,-29.291,-41.470,179.990,5.526,148.973
C01043=1205.914,-29.041,-41.483,179.993,5.526,148.972
C01044=1205.909,-28.791,-41.495,179.996,5.527,148.971
C01045=1205.903,-28.542,-41.509,179.998,5.526,148.971
C01046=1205.899,-28.292,-41.522,180.000,5.527,148.970
C01047=1205.894,-28.043,-41.534,-179.997,5.528,148.969
C01048=1205.889,-27.793,-41.547,-179.995,5.528,148.969
C01049=1205.883,-27.543,-41.560,-179.993,5.528,148.968
C01050=1205.878,-27.294,-41.573,-179.990,5.528,148.967
C01051=1205.873,-27.044,-41.586,-179.987,5.529,148.967
C01052=1205.869,-26.794,-41.598,-179.985,5.529,148.966
C01053=1205.863,-26.545,-41.612,-179.983,5.529,148.965
C01054=1205.858,-26.295,-41.624,-179.980,5.530,148.965
C01055=1205.853,-26.045,-41.637,-179.978,5.530,148.964
C01056=1205.847,-25.796,-41.650,-179.975,5.531,148.963
C01057=1205.842,-25.546,-41.663,-179.973,5.530,148.963
C01058=1205.838,-25.297,-41.677,-179.970,5.531,148.962
C01059=1205.832,-25.047,-41.690,-179.968,5.531,148.961
C01060=1205.827,-24.798,-41.703,-179.965,5.532,148.961
C01061=1205.822,-24.548,-41.715,-179.963,5.531,148.960
C01062=1205.816,-24.298,-41.729,-179.961,5.532,148.960
C01063=1205.812,-24.048,-41.742,-179.958,5.533,148.959
C01064=1205.807,-23.799,-41.754,-179.956,5.533,148.958
C01065=1205.801,-23.549,-41.767,-179.953,5.533,148.957
C01066=1205.796,-23.280,-41.782,-179.951,5.533,148.957
C01067=1205.791,-23.010,-41.796,-179.948,5.534,148.956
C01068=1205.785,-22.741,-41.809,-179.945,5.534,148.955
C01069=1205.779,-22.472,-41.824,-179.942,5.534,148.954
C01070=1205.775,-22.222,-41.837,-179.940,5.535,148.954
C01071=1205.769,-21.972,-41.851,-179.938,5.535,148.953
C01072=1205.764,-21.723,-41.863,-179.935,5.535,148.953
C01073=1205.759,-21.472,-41.877,-179.933,5.536,148.952
C01074=1205.754,-21.224,-41.890,-179.930,5.536,148.951
C01075=1205.749,-20.974,-41.903,-179.928,5.536,148.950
C01076=1205.744,-20.724,-41.916,-179.925,5.537,148.950
C01077=1205.738,-20.475,-41.929,-179.923,5.537,148.949
C01078=1205.733,-20.225,-41.943,-179.921,5.538,148.949
C01079=1205.728,-19.976,-41.956,-179.918,5.538,148.948
C01080=1205.723,-19.725,-41.969,-179.916,5.538,148.947
C01081=1205.718,-19.476,-41.982,-179.913,5.539,148.947
C01082=1205.714,-19.227,-41.996,-179.910,5.539,148.946
C01083=1205.708,-18.977,-42.009,-179.908,5.540,148.945
C01084=1205.703,-18.727,-42.022,-179.906,5.539,148.944
C01085=1205.698,-18.478,-42.036,-179.903,5.540,148.944
C01086=1205.693,-18.229,-42.048,-179.901,5.541,148.943
C01087=1205.687,-17.978,-42.062,-179.898,5.541,148.943
C01088=1205.683,-17.730,-42.075,-179.896,5.541,148.942
C01089=1205.677,-17.479,-42.089,-179.894,5.541,148.941
C01090=1205.672,-17.230,-42.101,-179.891,5.542,148.940
C01091=1205.667,-16.980,-42.116,-179.888,5.542,148.940
C01092=1205.662,-16.731,-42.128,-179.886,5.542,148.939
C01093=1205.657,-16.481,-42.142,-179.883,5.542,148.938
C01094=1205.652,-16.232,-42.155,-179.881,5.543,148.938
C01095=1205.647,-15.982,-42.169,-179.879,5.544,148.937
C01096=1205.642,-15.732,-42.181,-179.876,5.544,148.937
C01097=1205.637,-15.483,-42.195,-179.874,5.544,148.936
C01098=1205.632,-15.233,-42.208,-179.871,5.544,148.935
C01099=1205.627,-14.984,-42.222,-179.869,5.545,148.934
C01100=1205.621,-14.734,-42.236,-179.866,5.545,148.934
C01101=1205.617,-14.485,-42.249,-179.863,5.546,148.933
C01102=1205.611,-14.235,-42.262,-179.862,5.546,148.933
C01103=1205.606,-13.985,-42.275,-179.859,5.546,148.932
C01104=1205.601,-13.736,-42.289,-179.856,5.547,148.931
C01105=1205.596,-13.486,-42.302,-179.854,5.547,148.931
C01106=1205.591,-13.237,-42.316,-179.852,5.547,148.930
C01107=1205.585,-12.987,-42.330,-179.849,5.547,148.929
C01108=1205.581,-12.737,-42.343,-179.846,5.548,148.928
C01109=1205.575,-12.488,-42.357,-179.844,5.548,148.928
C01110=1205.571,-12.238,-42.370,-179.842,5.549,148.927
C01111=1205.565,-11.989,-42.383,-179.839,5.549,148.927
C01112=1205.560,-11.739,-42.398,-179.837,5.549,148.926
C01113=1205.555,-11.490,-42.410,-179.834,5.550,148.925
C01114=1205.550,-11.240,-42.425,-179.831,5.550,148.925
C01115=1205.545,-10.990,-42.437,-179.829,5.551,148.924
C01116=1205.540,-10.741,-42.452,-179.827,5.551,148.923
C01117=1205.535,-10.490,-42.465,-179.824,5.551,148.922
C01118=1205.530,-10.242,-42.478,-179.822,5.552,148.922
C01119=1205.525,-9.992,-42.493,-179.819,5.552,148.921
C01120=1205.519,-9.742,-42.506,-179.817,5.553,148.921
C01121=1205.515,-9.493,-42.520,-179.815,5.553,148.920
C01122=1205.510,-9.243,-42.533,-179.812,5.553,148.919
C01123=1205.504,-8.994,-42.547,-179.809,5.554,148.919
C01124=1205.500,-8.744,-42.561,-179.807,5.554,148.918
C01125=1205.494,-8.495,-42.574,-179.804,5.555,148.917
C01126=1205.489,-8.245,-42.588,-179.802,5.555,148.917
C01127=1205.485,-7.995,-42.601,-179.800,5.555,148.916
C01128=1205.479,-7.746,-42.615,-179.797,5.556,148.915
C01129=1205.474,-7.496,-42.629,-179.794,5.556,148.915
C01130=1205.468,-7.247,-42.643,-179.792,5.557,148.914
C01131=1205.464,-6.997,-42.656,-179.789,5.557,148.913
C01132=1205.459,-6.747,-42.670,-179.787,5.557,148.913
C01133=1205.453,-6.498,-42.684,-179.785,5.558,148.912
C01134=1205.449,-6.248,-42.697,-179.782,5.558,148.911
C01135=1205.444,-5.999,-42.712,-179.779,5.559,148.911
C01136=1205.438,-5.750,-42.726,-179.777,5.559,148.910
C01137=1205.433,-5.499,-42.739,-179.774,5.560,148.909
C01138=1205.429,-5.250,-42.753,-179.772,5.559,148.909
C01139=1205.423,-5.001,-42.767,-179.769,5.560,148.908
C01140=1205.418,-4.751,-42.780,-179.767,5.561,148.907
C01141=1205.413,-4.501,-42.795,-179.765,5.561,148.907
C01142=1205.408,-4.252,-42.808,-179.762,5.562,148.906
C01143=1205.403,-4.003,-42.822,-179.760,5.561,148.905
C01144=1205.398,-3.752,-42.836,-179.757,5.562,148.905
C01145=1205.393,-3.503,-42.850,-179.755,5.562,148.904
C01146=1205.388,-3.253,-42.864,-179.752,5.563,148.903
C01147=1205.383,-3.004,-42.878,-179.749,5.563,148.903
C01148=1205.378,-2.755,-42.891,-179.747,5.564,148.902
C01149=1205.373,-2.505,-42.905,-179.745,5.564,148.902
C01150=1205.368,-2.255,-42.919,-179.742,5.564,148.901
C01151=1205.362,-2.006,-42.933,-179.740,5.565,148.900
C01152=1205.357,-1.756,-42.948,-179.737,5.565,148.899
C01153=1205.352,-1.507,-42.962,-179.734,5.566,148.899
C01154=1205.348,-1.257,-42.975,-179.732,5.566,148.898
C01155=1205.342,-1.008,-42.989,-179.730,5.567,148.898
C01156=1205.337,-0.758,-43.003,-179.728,5.567,148.897
C01157=1205.332,-0.508,-43.017,-179.725,5.567,148.896
C01158=1205.327,-0.259,-43.031,-179.722,5.568,148.896
C01159=1205.322,-0.009,-43.045,-179.720,5.568,148.895
C01160=1205.317,0.240,-43.060,-179.717,5.569,148.894
C01161=1205.312,0.490,-43.074,-179.714,5.569,148.893
C01162=1205.307,0.739,-43.087,-179.713,5.569,148.893
C01163=1205.302,0.989,-43.101,-179.710,5.570,148.892
C01164=1205.297,1.239,-43.115,-179.707,5.570,148.892
C01165=1205.292,1.488,-43.129,-179.705,5.571,148.891
C01166=1205.286,1.737,-43.143,-179.702,5.571,148.890
C01167=1205.281,1.987,-43.158,-179.699,5.572,148.890
C01168=1205.276,2.237,-43.172,-179.697,5.572,148.889
C01169=1205.271,2.487,-43.186,-179.695,5.572,148.888
C01170=1205.266,2.755,-43.201,-179.692,5.573,148.887
C01171=1205.260,3.024,-43.216,-179.689,5.573,148.887
C01172=1205.255,3.294,-43.231,-179.687,5.574,148.886
C01173=1205.250,3.562,-43.247,-179.684,5.574,148.885
C01174=1205.245,3.812,-43.261,-179.681,5.575,148.885
C01175=1205.240,4.062,-43.276,-179.679,5.575,148.884
C01176=1205.234,4.311,-43.290,-179.677,5.576,148.884
C01177=1205.229,4.560,-43.304,-179.674,5.576,148.883
C01178=1205.224,4.810,-43.318,-179.671,5.577,148.882
C01179=1205.219,5.060,-43.332,-179.669,5.577,148.882
C01180=1205.214,5.310,-43.347,-179.666,5.578,148.881
C01181=1205.209,5.559,-43.361,-179.664,5.578,148.880
C01182=1205.204,5.808,-43.375,-179.662,5.579,148.880
C01183=1205.199,6.058,-43.389,-179.659,5.579,148.879
C01184=1205.194,6.308,-43.404,-179.656,5.580,148.878
C01185=1205.189,6.557,-43.418,-179.654,5.580,148.878
C01186=1205.184,6.807,-43.433,-179.651,5.581,148.877
C01187=1205.179,7.056,-43.447,-179.649,5.581,148.876
C01188=1205.174,7.305,-43.461,-179.646,5.582,148.876
C01189=1205.169,7.555,-43.475,-179.644,5.582,148.875
C01190=1205.164,7.805,-43.490,-179.642,5.582,148.874
C01191=1205.159,8.054,-43.504,-179.639,5.583,148.874
C01192=1205.154,8.304,-43.518,-179.636,5.583,148.873
C01193=1205.148,8.553,-43.532,-179.634,5.584,148.872
C01194=1205.143,8.802,-43.548,-179.631,5.584,148.872
C01195=1205.138,9.052,-43.562,-179.629,5.585,148.871
C01196=1205.133,9.302,-43.576,-179.626,5.586,148.871
C01197=1205.128,9.552,-43.590,-179.624,5.586,148.870
C01198=1205.123,9.801,-43.605,-179.621,5.586,148.869
C01199=1205.119,10.050,-43.620,-179.619,5.586,148.869
C01200=1205.114,10.300,-43.634,-179.616,5.587,148.868
C01201=1205.108,10.549,-43.648,-179.614,5.587,148.867
C01202=1205.103,10.799,-43.662,-179.611,5.588,148.867
C01203=1205.098,11.048,-43.677,-179.609,5.589,148.866
C01204=1205.093,11.298,-43.692,-179.606,5.589,148.865
C01205=1205.088,11.548,-43.706,-179.603,5.590,148.865
C01206=1205.083,11.797,-43.721,-179.601,5.590,148.864
C01207=1205.078,12.046,-43.736,-179.599,5.590,148.863
C01208=1205.073,12.296,-43.750,-179.597,5.591,148.863
C01209=1205.068,12.546,-43.764,-179.594,5.591,148.862
C01210=1205.063,12.796,-43.779,-179.591,5.592,148.861
C01211=1205.058,13.045,-43.794,-179.589,5.592,148.861
C01212=1205.052,13.294,-43.808,-179.586,5.593,148.860
C01213=1205.047,13.544,-43.822,-179.583,5.593,148.859
C01214=1205.043,13.793,-43.837,-179.581,5.594,148.859
C01215=1205.037,14.043,-43.852,-179.578,5.595,148.858
C01216=1205.032,14.293,-43.866,-179.576,5.595,148.858
C01217=1205.027,14.542,-43.881,-179.573,5.596,148.857
C01218=1205.023,14.791,-43.896,-179.571,5.595,148.856
C01219=1205.018,15.041,-43.910,-179.568,5.596,148.856
C01220=1205.012,15.290,-43.925,-179.566,5.597,148.855
C01221=1205.007,15.540,-43.940,-179.564,5.597,148.854
C01222=1205.003,15.789,-43.955,-179.561,5.598,148.854
C01223=1204.998,16.039,-43.969,-179.558,5.598,148.853
C01224=1204.992,16.289,-43.984,-179.556,5.599,148.852
C01225=1204.987,16.538,-43.999,-179.553,5.599,148.852
C01226=1204.982,16.788,-44.013,-179.551,5.600,148.851
C01227=1204.978,17.037,-44.028,-179.548,5.601,148.851
C01228=1204.972,17.287,-44.043,-179.546,5.601,148.850
C01229=1204.967,17.536,-44.058,-179.543,5.602,148.849
C01230=1204.962,17.786,-44.072,-179.540,5.602,148.848
C01231=1204.958,18.035,-44.087,-179.538,5.602,148.848
C01232=1204.952,18.285,-44.102,-179.536,5.603,148.847
C01233=1204.947,18.534,-44.117,-179.533,5.603,148.847
C01234=1204.942,18.784,-44.131,-179.531,5.604,148.846
C01235=1204.937,19.033,-44.147,-179.528,5.604,148.845
C01236=1204.932,19.283,-44.161,-179.525,5.605,148.845
C01237=1204.927,19.532,-44.176,-179.523,5.605,148.844
C01238=1204.922,19.782,-44.191,-179.521,5.606,148.843
C01239=1204.917,20.031,-44.206,-179.518,5.607,148.843
C01240=1204.912,20.281,-44.220,-179.515,5.607,148.842
C01241=1204.907,20.530,-44.236,-179.513,5.608,148.841
C01242=1204.902,20.780,-44.250,-179.510,5.608,148.841
C01243=1204.897,21.029,-44.265,-179.508,5.609,148.840
C01244=1204.891,21.279,-44.280,-179.505,5.610,148.840
C01245=1204.887,21.528,-44.295,-179.503,5.610,148.839
C01246=1204.881,21.777,-44.311,-179.500,5.611,148.838
C01247=1204.876,22.027,-44.325,-179.498,5.610,148.838
C01248=1204.872,22.276,-44.340,-179.495,5.611,148.837
C01249=1204.867,22.527,-44.355,-179.493,5.612,148.836
C01250=1204.862,22.776,-44.370,-179.490,5.612,148.836
C01251=1204.857,23.025,-44.385,-179.488,5.613,148.835
C01252=1204.852,23.275,-44.400,-179.485,5.613,148.834
C01253=1204.847,23.524,-44.415,-179.483,5.614,148.834
C01254=1204.842,23.774,-44.431,-179.480,5.615,148.833
C01255=1204.837,24.023,-44.445,-179.478,5.615,148.833
C01256=1204.831,24.273,-44.461,-179.475,5.616,148.832
C01257=1204.827,24.522,-44.476,-179.472,5.616,148.831
C01258=1204.822,24.772,-44.490,-179.470,5.617,148.831
C01259=1204.816,25.021,-44.505,-179.467,5.617,148.830
C01260=1204.812,25.271,-44.521,-179.465,5.618,148.829
C01261=1204.807,25.521,-44.536,-179.462,5.619,148.829
C01262=1204.802,25.770,-44.551,-179.460,5.619,148.828
C01263=1204.797,26.019,-44.566,-179.457,5.620,148.827
C01264=1204.792,26.268,-44.581,-179.454,5.620,148.827
C01265=1204.786,26.518,-44.596,-179.452,5.621,148.826
C01266=1204.782,26.767,-44.611,-179.450,5.622,148.826
C01267=1204.776,27.017,-44.627,-179.447,5.622,148.825
C01268=1204.772,27.267,-44.642,-179.444,5.623,148.824
C01269=1204.766,27.517,-44.657,-179.442,5.623,148.824
C01270=1204.762,27.766,-44.672,-179.440,5.624,148.823
C01271=1204.756,28.015,-44.687,-179.437,5.625,148.822
C01272=1204.752,28.264,-44.702,-179.434,5.625,148.822
C01273=1204.746,28.514,-44.718,-179.432,5.626,148.821
C01274=1204.741,28.783,-44.734,-179.429,5.626,148.820
C01275=1204.736,29.051,-44.751,-179.426,5.627,148.820
C01276=1204.730,29.321,-44.767,-179.424,5.627,148.819
C01277=1204.726,29.589,-44.784,-179.421,5.628,148.818
C01278=1204.720,29.838,-44.799,-179.418,5.628,148.818
C01279=1204.715,30.088,-44.814,-179.416,5.629,148.817
C01280=1204.710,30.337,-44.829,-179.414,5.630,148.817
C01281=1204.705,30.587,-44.845,-179.411,5.630,148.816
C01282=1204.700,30.837,-44.860,-179.408,5.631,148.815
C01283=1204.695,31.086,-44.876,-179.406,5.631,148.814
C01284=1204.690,31.335,-44.891,-179.403,5.632,148.814
C01285=1204.685,31.584,-44.906,-179.401,5.633,148.813
C01286=1204.680,31.834,-44.922,-179.398,5.633,148.813
C01287=1204.676,32.084,-44.937,-179.396,5.634,148.812
C01288=1204.670,32.333,-44.953,-179.393,5.634,148.811
C01289=1204.665,32.582,-44.969,-179.390,5.635,148.811
C01290=1204.660,32.832,-44.984,-179.388,5.636,148.810
C01291=1204.655,33.082,-44.999,-179.385,5.636,148.810
C01292=1204.650,33.331,-45.014,-179.383,5.637,148.809
C01293=1204.645,33.581,-45.029,-179.380,5.637,148.808
C01294=1204.640,33.830,-45.045,-179.378,5.638,148.808
C01295=1204.635,34.079,-45.060,-179.375,5.639,148.807
C01296=1204.630,34.329,-45.076,-179.373,5.639,148.806
C01297=1204.625,34.578,-45.092,-179.370,5.640,148.806
C01298=1204.621,34.827,-45.107,-179.367,5.640,148.805
C01299=1204.616,35.077,-45.123,-179.365,5.641,148.805
C01300=1204.610,35.327,-45.139,-179.363,5.642,148.804
C01301=1204.605,35.576,-45.154,-179.360,5.642,148.803
C01302=1204.600,35.825,-45.169,-179.357,5.643,148.803
C01303=1204.596,36.075,-45.185,-179.355,5.643,148.802
C01304=1204.590,36.325,-45.201,-179.353,5.644,148.801
C01305=1204.585,36.574,-45.216,-179.350,5.645,148.801
C01306=1204.580,36.823,-45.231,-179.347,5.645,148.800
C01307=1204.575,37.073,-45.247,-179.345,5.646,148.799
C01308=1204.570,37.323,-45.263,-179.343,5.647,148.799
C01309=1204.565,37.572,-45.278,-179.340,5.647,148.798
C01310=1204.561,37.821,-45.295,-179.337,5.648,148.798
C01311=1204.555,38.071,-45.310,-179.335,5.648,148.797
C01312=1204.550,38.320,-45.326,-179.332,5.649,148.796
C01313=1204.545,38.570,-45.342,-179.330,5.650,148.796
C01314=1204.541,38.819,-45.357,-179.327,5.650,148.795
C01315=1204.535,39.069,-45.372,-179.325,5.651,148.794
C01316=1204.530,39.319,-45.388,-179.322,5.651,148.794
C01317=1204.525,39.568,-45.405,-179.320,5.652,148.793
C01318=1204.521,39.817,-45.420,-179.317,5.653,148.793
C01319=1204.516,40.067,-45.436,-179.314,5.654,148.792
C01320=1204.511,40.316,-45.451,-179.311,5.655,148.791
C01321=1204.505,40.565,-45.467,-179.309,5.655,148.791
C01322=1204.501,40.815,-45.483,-179.306,5.656,148.790
C01323=1204.495,41.065,-45.499,-179.304,5.657,148.790
C01324=1204.491,41.314,-45.514,-179.301,5.657,148.789
C01325=1204.486,41.564,-45.530,-179.298,5.658,148.788
C01326=1204.481,41.812,-45.546,-179.296,5.659,148.788
C01327=1204.475,42.062,-45.562,-179.294,5.659,148.787
C01328=1204.471,42.312,-45.578,-179.291,5.660,148.786
C01329=1204.465,42.561,-45.594,-179.288,5.660,148.786
C01330=1204.461,42.811,-45.610,-179.286,5.661,148.785
C01331=1204.455,43.060,-45.626,-179.284,5.662,148.785
C01332=1204.451,43.309,-45.641,-179.281,5.662,148.784
C01333=1204.446,43.559,-45.657,-179.278,5.663,148.783
C01334=1204.441,43.808,-45.673,-179.276,5.663,148.783
C01335=1204.436,44.057,-45.689,-179.274,5.664,148.782
C01336=1204.431,44.307,-45.705,-179.271,5.665,148.781
C01337=1204.426,44.557,-45.721,-179.268,5.665,148.781
C01338=1204.421,44.806,-45.737,-179.266,5.666,148.780
C01339=1204.416,45.055,-45.753,-179.263,5.667,148.780
C01340=1204.411,45.306,-45.769,-179.260,5.668,148.779
C01341=1204.406,45.554,-45.785,-179.258,5.669,148.778
C01342=1204.400,45.804,-45.801,-179.255,5.669,148.778
C01343=1204.396,46.053,-45.817,-179.253,5.670,148.777
C01344=1204.391,46.303,-45.833,-179.250,5.670,148.777
C01345=1204.387,46.552,-45.848,-179.248,5.671,148.776
C01346=1204.381,46.801,-45.865,-179.245,5.672,148.775
C01347=1204.377,47.051,-45.881,-179.243,5.672,148.775
C01348=1204.372,47.300,-45.897,-179.240,5.673,148.774
C01349=1204.367,47.550,-45.913,-179.238,5.674,148.773
C01350=1204.362,47.799,-45.929,-179.235,5.674,148.773
C01351=1204.356,48.048,-45.945,-179.233,5.675,148.772
C01352=1204.352,48.298,-45.961,-179.230,5.676,148.772
C01353=1204.346,48.547,-45.977,-179.227,5.677,148.771
C01354=1204.342,48.797,-45.994,-179.224,5.677,148.770
C01355=1204.337,49.046,-46.009,-179.222,5.678,148.770
C01356=1204.332,49.296,-46.026,-179.219,5.679,148.769
C01357=1204.326,49.545,-46.042,-179.217,5.679,148.769
C01358=1204.321,49.795,-46.059,-179.214,5.680,148.768
C01359=1204.316,50.044,-46.074,-179.212,5.681,148.767
C01360=1204.312,50.294,-46.091,-179.209,5.681,148.767
C01361=1204.307,50.542,-46.107,-179.207,5.682,148.766
C01362=1204.302,50.793,-46.123,-179.204,5.682,148.765
C01363=1204.297,51.041,-46.140,-179.202,5.683,148.765
C01364=1204.292,51.291,-46.156,-179.199,5.684,148.764
C01365=1204.287,51.540,-46.172,-179.196,5.685,148.764
C01366=1204.282,51.790,-46.189,-179.193,5.686,148.763
C01367=1204.278,52.040,-46.205,-179.191,5.687,148.763
C01368=1204.272,52.289,-46.221,-179.189,5.687,148.762
C01369=1204.268,52.539,-46.237,-179.186,5.688,148.761
C01370=1204.263,52.788,-46.253,-179.184,5.689,148.761
C01371=1204.257,53.037,-46.270,-179.181,5.689,148.760
C01372=1204.252,53.287,-46.286,-179.179,5.690,148.759
C01373=1204.248,53.536,-46.303,-179.176,5.690,148.759
C01374=1204.242,53.785,-46.319,-179.174,5.691,148.758
C01375=1204.238,54.035,-46.335,-179.171,5.693,148.758
C01376=1204.233,54.284,-46.351,-179.168,5.693,148.757
C01377=1204.228,54.533,-46.368,-179.165,5.694,148.756
C01378=1204.222,54.802,-46.385,-179.163,5.695,148.756
C01379=1204.217,55.071,-46.404,-179.161,5.695,148.755
C01380=1204.212,55.339,-46.421,-179.157,5.696,148.755
C01381=1204.207,55.608,-46.439,-179.155,5.697,148.754
C01382=1204.201,55.857,-46.456,-179.152,5.698,148.753
C01383=1204.196,56.107,-46.472,-179.149,5.698,148.753
C01384=1204.191,56.356,-46.488,-179.147,5.699,148.752
C01385=1204.187,56.605,-46.505,-179.145,5.700,148.751
C01386=1204.182,56.855,-46.521,-179.141,5.701,148.751
C01387=1204.176,57.104,-46.538,-179.139,5.701,148.750
C01388=1204.172,57.354,-46.554,-179.137,5.702,148.750
C01389=1204.167,57.603,-46.570,-179.134,5.703,148.749
C01390=1204.162,57.852,-46.587,-179.131,5.703,148.748
C01391=1204.157,58.102,-46.604,-179.129,5.704,148.748
C01392=1204.152,58.351,-46.621,-179.127,5.705,148.747
C01393=1204.147,58.600,-46.637,-179.124,5.705,148.747
C01394=1204.143,58.850,-46.653,-179.121,5.707,148.746
C01395=1204.137,59.099,-46.670,-179.119,5.708,148.746
C01396=1204.132,59.349,-46.687,-179.116,5.708,148.745
C01397=1204.127,59.598,-46.703,-179.113,5.709,148.744
C01398=1204.122,59.847,-46.720,-179.111,5.710,148.744
C01399=1204.117,60.097,-46.737,-179.109,5.710,148.743
C01400=1204.112,60.346,-46.753,-179.106,5.711,148.742
C01401=1204.108,60.595,-46.770,-179.103,5.712,148.742
C01402=1204.103,60.845,-46.787,-179.101,5.713,148.741
C01403=1204.098,61.094,-46.804,-179.098,5.714,148.741
C01404=1204.093,61.343,-46.820,-179.095,5.714,148.740
C01405=1204.088,61.594,-46.837,-179.093,5.715,148.740
C01406=1204.083,61.843,-46.853,-179.091,5.716,148.739
C01407=1204.078,62.092,-46.870,-179.088,5.716,148.738
C01408=1204.073,62.342,-46.887,-179.085,5.718,148.738
C01409=1204.068,62.591,-46.904,-179.083,5.718,148.737
C01410=1204.063,62.840,-46.920,-179.080,5.719,148.736
C01411=1204.058,63.090,-46.937,-179.077,5.720,148.736
C01412=1204.054,63.339,-46.954,-179.075,5.720,148.735
C01413=1204.048,63.588,-46.971,-179.073,5.721,148.735
C01414=1204.043,63.838,-46.987,-179.069,5.722,148.734
C01415=1204.039,64.087,-47.005,-179.067,5.723,148.734
C01416=1204.034,64.337,-47.022,-179.065,5.724,148.733
C01417=1204.029,64.585,-47.038,-179.062,5.724,148.732
C01418=1204.024,64.835,-47.056,-179.060,5.725,148.732
C01419=1204.019,65.085,-47.072,-179.057,5.726,148.731
C01420=1204.015,65.334,-47.089,-179.054,5.727,148.731
C01421=1204.009,65.583,-47.106,-179.052,5.728,148.730
C01422=1204.004,65.833,-47.123,-179.049,5.729,148.729
C01423=1203.999,66.082,-47.140,-179.047,5.729,148.729
C01424=1203.995,66.332,-47.157,-179.044,5.730,148.728
C01425=1203.989,66.581,-47.173,-179.042,5.731,148.728
C01426=1203.985,66.830,-47.191,-179.039,5.732,148.727
C01427=1203.979,67.080,-47.208,-179.036,5.733,148.726
C01428=1203.975,67.329,-47.225,-179.034,5.734,148.726
C01429=1203.970,67.578,-47.241,-179.031,5.734,148.725
C01430=1203.965,67.828,-47.258,-179.029,5.735,148.725
C01431=1203.960,68.077,-47.275,-179.026,5.736,148.724
C01432=1203.955,68.326,-47.293,-179.023,5.737,148.724
C01433=1203.951,68.576,-47.310,-179.021,5.737,148.723
C01434=1203.945,68.825,-47.327,-179.018,5.738,148.722
C01435=1203.940,69.075,-47.343,-179.016,5.739,148.722
C01436=1203.936,69.324,-47.361,-179.013,5.740,148.721
C01437=1203.930,69.573,-47.378,-179.010,5.741,148.721
C01438=1203.926,69.823,-47.395,-179.008,5.742,148.720
C01439=1203.920,70.072,-47.412,-179.005,5.742,148.719
C01440=1203.916,70.321,-47.429,-179.003,5.743,148.719
C01441=1203.911,70.571,-47.447,-179.000,5.744,148.718
C01442=1203.906,70.820,-47.463,-178.997,5.745,148.718
C01443=1203.901,71.070,-47.481,-178.995,5.746,148.717
C01444=1203.897,71.319,-47.498,-178.992,5.747,148.717
C01445=1203.891,71.568,-47.515,-178.990,5.747,148.716
C01446=1203.886,71.818,-47.532,-178.988,5.748,148.715
C01447=1203.882,72.067,-47.550,-178.984,5.750,148.715
C01448=1203.876,72.316,-47.567,-178.982,5.750,148.714
C01449=1203.872,72.566,-47.583,-178.980,5.751,148.714
C01450=1203.867,72.815,-47.601,-178.977,5.752,148.713
C01451=1203.862,73.065,-47.619,-178.974,5.752,148.712
C01452=1203.857,73.314,-47.635,-178.972,5.754,148.712
C01453=1203.852,73.563,-47.653,-178.969,5.754,148.711
C01454=1203.847,73.812,-47.670,-178.967,5.755,148.711
C01455=1203.842,74.061,-47.688,-178.964,5.756,148.710
C01456=1203.837,74.311,-47.705,-178.961,5.757,148.710
C01457=1203.833,74.561,-47.722,-178.959,5.758,148.709
C01458=1203.828,74.810,-47.740,-178.956,5.759,148.708
C01459=1203.823,75.060,-47.757,-178.954,5.759,148.708
C01460=1203.818,75.309,-47.774,-178.952,5.760,148.707
C01461=1203.813,75.558,-47.791,-178.948,5.762,148.707
C01462=1203.808,75.807,-47.809,-178.946,5.762,148.706
C01463=1203.803,76.056,-47.826,-178.944,5.763,148.706
C01464=1203.798,76.306,-47.844,-178.941,5.764,148.705
C01465=1203.793,76.555,-47.861,-178.938,5.765,148.704
C01466=1203.788,76.804,-47.879,-178.936,5.766,148.704
C01467=1203.784,77.054,-47.896,-178.933,5.766,148.703
C01468=1203.779,77.303,-47.914,-178.930,5.767,148.703
C01469=1203.773,77.553,-47.931,-178.928,5.769,148.702
C01470=1203.769,77.802,-47.949,-178.925,5.769,148.701
C01471=1203.764,78.052,-47.966,-178.923,5.770,148.701
C01472=1203.759,78.301,-47.984,-178.920,5.771,148.700
C01473=1203.754,78.551,-48.001,-178.918,5.771,148.700
C01474=1203.749,78.800,-48.019,-178.915,5.773,148.699
C01475=1203.745,79.049,-48.036,-178.912,5.774,148.699
C01476=1203.740,79.298,-48.053,-178.910,5.774,148.698
C01477=1203.735,79.548,-48.071,-178.908,5.775,148.698
C01478=1203.730,79.797,-48.089,-178.904,5.777,148.697
C01479=1203.725,80.046,-48.106,-178.902,5.777,148.697
C01480=1203.720,80.295,-48.124,-178.900,5.778,148.696
C01481=1203.715,80.545,-48.141,-178.897,5.779,148.695
C01482=1203.710,80.813,-48.160,-178.894,5.780,148.695
C01483=1203.704,81.082,-48.179,-178.892,5.781,148.694
C01484=1203.699,81.350,-48.198,-178.888,5.782,148.693
C01485=1203.694,81.618,-48.218,-178.886,5.783,148.693
C01486=1203.689,81.868,-48.235,-178.883,5.783,148.692
C01487=1203.685,82.117,-48.252,-178.880,5.785,148.692
C01488=1203.680,82.366,-48.270,-178.878,5.786,148.691
C01489=1203.674,82.616,-48.288,-178.876,5.787,148.691
C01490=1203.670,82.865,-48.306,-178.873,5.788,148.690
C01491=1203.665,83.114,-48.324,-178.870,5.789,148.689
C01492=1203.660,83.363,-48.342,-178.868,5.790,148.689
C01493=1203.655,83.613,-48.359,-178.865,5.790,148.688
C01494=1203.650,83.862,-48.377,-178.862,5.792,148.688
C01495=1203.645,84.111,-48.394,-178.860,5.792,148.687
C01496=1203.641,84.360,-48.412,-178.857,5.793,148.687
C01497=1203.635,84.610,-48.430,-178.855,5.794,148.686
C01498=1203.630,84.859,-48.448,-178.852,5.795,148.685
C01499=1203.625,85.108,-48.465,-178.849,5.796,148.685
C01500=1203.621,85.358,-48.483,-178.847,5.797,148.684
C01501=1203.616,85.608,-48.502,-178.844,5.798,148.684
C01502=1203.611,85.857,-48.519,-178.842,5.799,148.683
C01503=1203.606,86.106,-48.537,-178.839,5.800,148.683
C01504=1203.601,86.356,-48.555,-178.836,5.800,148.682
C01505=1203.596,86.605,-48.573,-178.834,5.802,148.682
C01506=1203.591,86.854,-48.591,-178.831,5.803,148.681
C01507=1203.586,87.103,-48.609,-178.829,5.803,148.681
C01508=1203.582,87.352,-48.627,-178.826,5.805,148.680
C01509=1203.577,87.602,-48.645,-178.824,5.806,148.679
C01510=1203.571,87.851,-48.662,-178.821,5.806,148.679
C01511=1203.567,88.101,-48.680,-178.818,5.807,148.678
C01512=1203.562,88.350,-48.699,-178.816,5.809,148.678
C01513=1203.557,88.600,-48.717,-178.813,5.809,148.677
C01514=1203.552,88.849,-48.734,-178.811,5.810,148.677
C01515=1203.547,89.098,-48.752,-178.808,5.812,148.676
C01516=1203.543,89.347,-48.770,-178.805,5.812,148.675
C01517=1203.538,89.596,-48.788,-178.803,5.813,148.675
C01518=1203.533,89.845,-48.806,-178.800,5.814,148.674
C01519=1203.528,90.095,-48.825,-178.798,5.815,148.674
C01520=1203.524,90.345,-48.843,-178.795,5.816,148.673
C01521=1203.519,90.594,-48.861,-178.792,5.817,148.673
C01522=1203.514,90.843,-48.879,-178.790,5.818,148.672
C01523=1203.509,91.092,-48.897,-178.787,5.819,148.672
C01524=1203.504,91.341,-48.915,-178.785,5.820,148.671
C01525=1203.499,91.590,-48.933,-178.782,5.821,148.670
C01526=1203.495,91.840,-48.951,-178.780,5.822,148.670
C01527=1203.490,92.089,-48.969,-178.777,5.823,148.669
C01528=1203.484,92.339,-48.988,-178.774,5.824,148.669
C01529=1203.479,92.588,-49.006,-178.772,5.825,148.668
C01530=1203.475,92.837,-49.024,-178.769,5.826,148.668
C01531=1203.470,93.087,-49.043,-178.766,5.827,148.667
C01532=1203.465,93.336,-49.061,-178.764,5.828,148.667
C01533=1203.460,93.585,-49.079,-178.762,5.829,148.666
C01534=1203.456,93.834,-49.096,-178.758,5.830,148.666
C01535=1203.451,94.083,-49.114,-178.756,5.831,148.665
C01536=1203.446,94.333,-49.133,-178.754,5.832,148.664
C01537=1203.441,94.583,-49.151,-178.751,5.833,148.664
C01538=1203.436,94.831,-49.170,-178.748,5.834,148.663
C01539=1203.431,95.080,-49.188,-178.746,5.835,148.663
C01540=1203.427,95.330,-49.206,-178.743,5.836,148.662
C01541=1203.421,95.580,-49.225,-178.740,5.837,148.662
C01542=1203.416,95.829,-49.243,-178.738,5.838,148.661
C01543=1203.412,96.077,-49.262,-178.735,5.839,148.661
C01544=1203.407,96.327,-49.280,-178.733,5.840,148.660
C01545=1203.402,96.576,-49.298,-178.730,5.841,148.660
C01546=1203.397,96.826,-49.317,-178.727,5.842,148.659
C01547=1203.392,97.075,-49.335,-178.725,5.843,148.659
C01548=1203.388,97.324,-49.354,-178.722,5.845,148.658
C01549=1203.383,97.574,-49.372,-178.720,5.845,148.657
C01550=1203.377,97.823,-49.390,-178.717,5.846,148.657
C01551=1203.373,98.072,-49.409,-178.714,5.848,148.656
C01552=1203.368,98.321,-49.427,-178.712,5.848,148.656
C01553=1203.363,98.571,-49.445,-178.710,5.849,148.655
C01554=1203.358,98.820,-49.464,-178.706,5.851,148.655
C01555=1203.354,99.069,-49.483,-178.704,5.852,148.654
C01556=1203.349,99.319,-49.501,-178.702,5.852,148.654
C01557=1203.344,99.567,-49.520,-178.699,5.854,148.653
C01558=1203.339,99.817,-49.538,-178.696,5.855,148.653
C01559=1203.334,100.067,-49.556,-178.694,5.855,148.652
C01560=1203.330,100.315,-49.575,-178.691,5.857,148.652
C01561=1203.324,100.565,-49.594,-178.688,5.857,148.651
C01562=1203.320,100.814,-49.612,-178.686,5.859,148.650
C01563=1203.315,101.063,-49.631,-178.683,5.860,148.650
C01564=1203.310,101.312,-49.649,-178.681,5.861,148.649
C01565=1203.305,101.562,-49.668,-178.678,5.862,148.649
C01566=1203.301,101.811,-49.686,-178.676,5.863,148.648
C01567=1203.295,102.060,-49.706,-178.673,5.864,148.648
C01568=1203.291,102.310,-49.724,-178.670,5.865,148.647
C01569=1203.286,102.559,-49.743,-178.668,5.866,148.647
C01570=1203.281,102.808,-49.762,-178.665,5.868,148.646
C01571=1203.276,103.058,-49.780,-178.662,5.868,148.646
C01572=1203.271,103.306,-49.799,-178.660,5.869,148.645
C01573=1203.267,103.556,-49.817,-178.657,5.871,148.645
C01574=1203.261,103.805,-49.837,-178.655,5.872,148.644
C01575=1203.256,104.054,-49.855,-178.652,5.873,148.644
C01576=1203.252,104.304,-49.874,-178.650,5.874,148.643
C01577=1203.247,104.552,-49.893,-178.647,5.875,148.642
C01578=1203.243,104.802,-49.911,-178.644,5.876,148.642
C01579=1203.237,105.051,-49.930,-178.642,5.877,148.641
C01580=1203.233,105.300,-49.948,-178.639,5.879,148.641
C01581=1203.228,105.550,-49.968,-178.636,5.879,148.640
C01582=1203.223,105.799,-49.986,-178.634,5.880,148.640
C01583=1203.219,106.048,-50.005,-178.631,5.882,148.639
C01584=1203.214,106.297,-50.024,-178.629,5.882,148.639
C01585=1203.209,106.546,-50.042,-178.626,5.884,148.638
C01586=1203.204,106.815,-50.064,-178.623,5.884,148.638
C01587=1203.198,107.084,-50.084,-178.620,5.886,148.637
C01588=1203.193,107.352,-50.105,-178.618,5.887,148.637
C01589=1203.188,107.621,-50.124,-178.615,5.888,148.636
C01590=1203.183,107.869,-50.143,-178.613,5.889,148.636
C01591=1203.179,108.119,-50.162,-178.609,5.891,148.635
C01592=1203.173,108.368,-50.181,-178.607,5.891,148.634
C01593=1203.169,108.617,-50.200,-178.604,5.893,148.634
C01594=1203.164,108.866,-50.219,-178.602,5.894,148.633
C01595=1203.159,109.116,-50.238,-178.599,5.894,148.633
C01596=1203.154,109.365,-50.257,-178.597,5.896,148.632
C01597=1203.150,109.614,-50.276,-178.594,5.897,148.632
C01598=1203.145,109.863,-50.295,-178.591,5.899,148.631
C01599=1203.139,110.113,-50.314,-178.589,5.899,148.631
C01600=1203.135,110.362,-50.333,-178.586,5.901,148.630
C01601=1203.130,110.611,-50.353,-178.584,5.902,148.630
C01602=1203.126,110.860,-50.371,-178.581,5.902,148.629
C01603=1203.120,111.110,-50.390,-178.579,5.904,148.629
C01604=1203.115,111.359,-50.410,-178.576,5.905,148.628
C01605=1203.111,111.608,-50.429,-178.573,5.907,148.628
C01606=1203.106,111.857,-50.448,-178.571,5.907,148.627
C01607=1203.102,112.106,-50.467,-178.568,5.909,148.627
C01608=1203.096,112.356,-50.485,-178.565,5.909,148.626
C01609=1203.091,112.606,-50.505,-178.563,5.911,148.626
C01610=1203.087,112.854,-50.524,-178.560,5.912,148.625
C01611=1203.082,113.104,-50.544,-178.558,5.913,148.625
C01612=1203.077,113.353,-50.563,-178.555,5.914,148.624
C01613=1203.073,113.602,-50.582,-178.553,5.915,148.624
C01614=1203.067,113.851,-50.601,-178.549,5.917,148.623
C01615=1203.063,114.100,-50.621,-178.547,5.917,148.623
C01616=1203.058,114.349,-50.639,-178.545,5.919,148.622
C01617=1203.053,114.599,-50.658,-178.542,5.920,148.622
C01618=1203.048,114.849,-50.678,-178.539,5.922,148.621
C01619=1203.043,115.097,-50.697,-178.537,5.922,148.621
C01620=1203.039,115.347,-50.716,-178.534,5.924,148.620
C01621=1203.034,115.596,-50.736,-178.531,5.925,148.619
C01622=1203.029,115.845,-50.755,-178.529,5.925,148.619
C01623=1203.024,116.094,-50.774,-178.526,5.927,148.618
C01624=1203.019,116.343,-50.794,-178.524,5.928,148.618
C01625=1203.015,116.593,-50.813,-178.521,5.929,148.617
C01626=1203.009,116.842,-50.833,-178.519,5.930,148.617
C01627=1203.005,117.091,-50.852,-178.516,5.932,148.617
C01628=1203.000,117.340,-50.871,-178.513,5.933,148.616
C01629=1202.995,117.589,-50.891,-178.511,5.934,148.616
C01630=1202.991,117.839,-50.910,-178.508,5.935,148.615
C01631=1202.985,118.088,-50.930,-178.505,5.937,148.615
C01632=1202.981,118.337,-50.949,-178.503,5.937,148.614
C01633=1202.976,118.586,-50.968,-178.500,5.939,148.613
C01634=1202.971,118.835,-50.988,-178.498,5.940,148.613
C01635=1202.967,119.084,-51.008,-178.495,5.941,148.612
C01636=1202.961,119.333,-51.027,-178.493,5.942,148.612
C01637=1202.957,119.583,-51.046,-178.489,5.944,148.611
C01638=1202.953,119.832,-51.066,-178.487,5.945,148.611
C01639=1202.947,120.081,-51.085,-178.484,5.946,148.610
C01640=1202.942,120.331,-51.105,-178.482,5.947,148.610
C01641=1202.938,120.580,-51.125,-178.479,5.949,148.610
C01642=1202.933,120.828,-51.145,-178.477,5.949,148.609
C01643=1202.929,121.078,-51.164,-178.474,5.951,148.609
C01644=1202.924,121.327,-51.183,-178.471,5.952,148.608
C01645=1202.919,121.576,-51.203,-178.469,5.954,148.608
C01646=1202.914,121.826,-51.222,-178.466,5.954,148.607
C01647=1202.909,122.075,-51.243,-178.463,5.956,148.606
C01648=1202.904,122.323,-51.262,-178.461,5.957,148.606
C01649=1202.899,122.573,-51.282,-178.458,5.958,148.605
C01650=1202.895,122.823,-51.301,-178.456,5.959,148.605
C01651=1202.889,123.071,-51.321,-178.453,5.961,148.604
C01652=1202.885,123.320,-51.341,-178.451,5.962,148.604
C01653=1202.881,123.570,-51.360,-178.448,5.963,148.604
C01654=1202.876,123.819,-51.380,-178.445,5.964,148.603
C01655=1202.871,124.067,-51.400,-178.443,5.966,148.603
C01656=1202.866,124.317,-51.419,-178.440,5.966,148.602
C01657=1202.862,124.567,-51.439,-178.437,5.968,148.602
C01658=1202.857,124.816,-51.459,-178.435,5.969,148.601
C01659=1202.852,125.064,-51.479,-178.432,5.971,148.601
C01660=1202.847,125.314,-51.498,-178.430,5.971,148.600
C01661=1202.843,125.563,-51.519,-178.427,5.973,148.600
C01662=1202.838,125.812,-51.538,-178.425,5.974,148.599
C01663=1202.832,126.061,-51.558,-178.422,5.976,148.599
C01664=1202.828,126.310,-51.578,-178.419,5.976,148.598
C01665=1202.823,126.560,-51.598,-178.417,5.978,148.598
C01666=1202.819,126.809,-51.617,-178.414,5.979,148.597
C01667=1202.814,127.058,-51.637,-178.411,5.980,148.597
C01668=1202.809,127.307,-51.657,-178.409,5.981,148.596
C01669=1202.804,127.556,-51.677,-178.406,5.983,148.596
C01670=1202.800,127.806,-51.697,-178.403,5.984,148.595
C01671=1202.795,128.054,-51.717,-178.401,5.985,148.595
C01672=1202.790,128.304,-51.737,-178.398,5.987,148.594
C01673=1202.785,128.553,-51.757,-178.396,5.988,148.594
C01674=1202.780,128.802,-51.777,-178.393,5.989,148.593
C01675=1202.775,129.051,-51.798,-178.391,5.990,148.593
C01676=1202.771,129.301,-51.817,-178.388,5.992,148.592
C01677=1202.766,129.549,-51.837,-178.385,5.993,148.592
C01678=1202.761,129.799,-51.857,-178.383,5.994,148.591
C01679=1202.756,130.048,-51.877,-178.380,5.995,148.591
C01680=1202.752,130.297,-51.897,-178.377,5.997,148.590
C01681=1202.747,130.546,-51.917,-178.375,5.998,148.590
C01682=1202.742,130.795,-51.937,-178.372,5.999,148.589
C01683=1202.737,131.044,-51.958,-178.369,6.001,148.589
C01684=1202.732,131.294,-51.977,-178.367,6.002,148.589
C01685=1202.728,131.543,-51.998,-178.364,6.003,148.588
C01686=1202.723,131.792,-52.018,-178.362,6.004,148.588
C01687=1202.718,132.041,-52.038,-178.359,6.006,148.587
C01688=1202.714,132.290,-52.058,-178.357,6.007,148.587
C01689=1202.709,132.539,-52.077,-178.354,6.008,148.586
C01690=1202.703,132.808,-52.100,-178.351,6.010,148.586
C01691=1202.698,133.077,-52.122,-178.348,6.012,148.585
C01692=1202.694,133.345,-52.144,-178.346,6.012,148.584
C01693=1202.688,133.614,-52.165,-178.343,6.014,148.584
C01694=1202.684,133.863,-52.186,-178.340,6.015,148.583
C01695=1202.679,134.112,-52.206,-178.338,6.016,148.583
C01696=1202.674,134.361,-52.225,-178.335,6.018,148.583
C01697=1202.669,134.610,-52.246,-178.332,6.019,148.582
C01698=1202.664,134.859,-52.267,-178.330,6.021,148.582
C01699=1202.659,135.109,-52.286,-178.327,6.022,148.581
C01700=1202.655,135.358,-52.307,-178.324,6.023,148.581
C01701=1202.650,135.607,-52.328,-178.322,6.025,148.580
C01702=1202.645,135.856,-52.348,-178.320,6.026,148.580
C01703=1202.641,136.105,-52.368,-178.316,6.027,148.579
C01704=1202.636,136.354,-52.388,-178.314,6.029,148.579
C01705=1202.631,136.604,-52.409,-178.312,6.030,148.578
C01706=1202.627,136.853,-52.429,-178.308,6.031,148.578
C01707=1202.622,137.102,-52.450,-178.306,6.032,148.577
C01708=1202.617,137.351,-52.470,-178.304,6.034,148.577
C01709=1202.612,137.600,-52.490,-178.300,6.035,148.576
C01710=1202.608,137.849,-52.511,-178.298,6.036,148.576
C01711=1202.602,138.098,-52.531,-178.296,6.038,148.576
C01712=1202.598,138.347,-52.552,-178.293,6.039,148.575
C01713=1202.593,138.596,-52.572,-178.290,6.041,148.575
C01714=1202.588,138.845,-52.593,-178.288,6.042,148.574
C01715=1202.583,139.095,-52.613,-178.285,6.043,148.574
C01716=1202.579,139.344,-52.633,-178.282,6.045,148.573
C01717=1202.574,139.593,-52.654,-178.280,6.046,148.573
C01718=1202.569,139.842,-52.674,-178.278,6.047,148.572
C01719=1202.565,140.091,-52.695,-178.274,6.049,148.572
C01720=1202.560,140.340,-52.716,-178.272,6.050,148.571
C01721=1202.555,140.589,-52.736,-178.270,6.052,148.571
C01722=1202.550,140.838,-52.757,-178.267,6.052,148.570
C01723=1202.546,141.087,-52.777,-178.264,6.054,148.570
C01724=1202.541,141.336,-52.798,-178.262,6.056,148.570
C01725=1202.536,141.585,-52.819,-178.259,6.056,148.569
C01726=1202.531,141.834,-52.839,-178.256,6.058,148.569
C01727=1202.527,142.084,-52.861,-178.254,6.060,148.568
C01728=1202.522,142.333,-52.881,-178.251,6.061,148.568
C01729=1202.517,142.582,-52.902,-178.248,6.062,148.567
C01730=1202.513,142.831,-52.922,-178.246,6.063,148.567
C01731=1202.508,143.081,-52.943,-178.244,6.065,148.567
C01732=1202.503,143.330,-52.964,-178.241,6.067,148.566
C01733=1202.499,143.579,-52.984,-178.238,6.067,148.566
C01734=1202.494,143.828,-53.005,-178.236,6.069,148.565
C01735=1202.489,144.077,-53.025,-178.233,6.071,148.565
C01736=1202.484,144.326,-53.046,-178.230,6.072,148.564
C01737=1202.480,144.574,-53.067,-178.228,6.073,148.564
C01738=1202.475,144.824,-53.088,-178.225,6.075,148.563
C01739=1202.470,145.073,-53.109,-178.222,6.076,148.563
C01740=1202.465,145.322,-53.130,-178.220,6.078,148.562
C01741=1202.460,145.571,-53.151,-178.217,6.079,148.562
C01742=1202.456,145.821,-53.171,-178.215,6.080,148.561
C01743=1202.451,146.070,-53.192,-178.212,6.082,148.561
C01744=1202.447,146.318,-53.213,-178.209,6.084,148.561
C01745=1202.442,146.568,-53.234,-178.207,6.085,148.560
C01746=1202.437,146.817,-53.255,-178.204,6.086,148.560
C01747=1202.432,147.066,-53.276,-178.201,6.088,148.559
C01748=1202.428,147.314,-53.297,-178.199,6.089,148.559
C01749=1202.423,147.563,-53.318,-178.196,6.091,148.558
C01750=1202.418,147.813,-53.339,-178.194,6.091,148.558
C01751=1202.414,148.062,-53.359,-178.191,6.093,148.557
C01752=1202.409,148.311,-53.381,-178.188,6.095,148.557
C01753=1202.404,148.560,-53.402,-178.186,6.097,148.557
C01754=1202.399,148.809,-53.422,-178.183,6.097,148.556
C01755=1202.394,149.058,-53.443,-178.181,6.099,148.556
C01756=1202.390,149.307,-53.465,-178.178,6.101,148.555
C01757=1202.385,149.557,-53.486,-178.176,6.102,148.555
C01758=1202.380,149.806,-53.507,-178.173,6.103,148.554
C01759=1202.376,150.054,-53.528,-178.170,6.105,148.554
C01760=1202.371,150.304,-53.549,-178.168,6.106,148.554
C01761=1202.366,150.553,-53.570,-178.165,6.108,148.553
C01762=1202.362,150.801,-53.591,-178.162,6.109,148.553
C01763=1202.357,151.051,-53.612,-178.160,6.110,148.552
C01764=1202.352,151.300,-53.633,-178.157,6.112,148.552
C01765=1202.348,151.549,-53.654,-178.154,6.114,148.551
C01766=1202.342,151.798,-53.675,-178.152,6.114,148.551
C01767=1202.338,152.047,-53.697,-178.149,6.116,148.550
C01768=1202.333,152.297,-53.718,-178.147,6.118,148.550
C01769=1202.329,152.545,-53.739,-178.144,6.119,148.550
C01770=1202.324,152.794,-53.760,-178.141,6.120,148.549
C01771=1202.319,153.043,-53.781,-178.139,6.122,148.549
C01772=1202.314,153.293,-53.803,-178.136,6.124,148.548
C01773=1202.310,153.542,-53.824,-178.134,6.125,148.548
C01774=1202.305,153.790,-53.845,-178.131,6.126,148.547
C01775=1202.300,154.040,-53.866,-178.128,6.128,148.547
C01776=1202.296,154.289,-53.888,-178.126,6.129,148.547
C01777=1202.291,154.538,-53.909,-178.123,6.131,148.546
C01778=1202.286,154.787,-53.931,-178.121,6.133,148.546
C01779=1202.281,155.035,-53.952,-178.117,6.134,148.545
C01780=1202.277,155.285,-53.974,-178.115,6.135,148.545
C01781=1202.272,155.534,-53.995,-178.113,6.137,148.544
C01782=1202.267,155.783,-54.016,-178.110,6.139,148.544
C01783=1202.263,156.031,-54.037,-178.108,6.140,148.544
C01784=1202.258,156.281,-54.059,-178.105,6.141,148.543
C01785=1202.253,156.530,-54.080,-178.102,6.143,148.543
C01786=1202.248,156.779,-54.102,-178.099,6.145,148.542
C01787=1202.244,157.029,-54.123,-178.097,6.146,148.542
C01788=1202.239,157.277,-54.145,-178.095,6.147,148.542
C01789=1202.235,157.526,-54.166,-178.091,6.149,148.541
C01790=1202.230,157.775,-54.187,-178.089,6.150,148.541
C01791=1202.225,158.024,-54.209,-178.087,6.152,148.540
C01792=1202.220,158.273,-54.231,-178.084,6.153,148.540
C01793=1202.215,158.522,-54.252,-178.081,6.155,148.539
C01794=1202.210,158.791,-54.274,-178.078,6.157,148.539
C01795=1202.205,159.060,-54.299,-178.075,6.158,148.538
C01796=1202.200,159.329,-54.322,-178.072,6.160,148.538
C01797=1202.195,159.598,-54.345,-178.070,6.161,148.537
C01798=1202.191,159.848,-54.367,-178.067,6.163,148.537
C01799=1202.186,160.096,-54.388,-178.065,6.164,148.537
C01800=1202.181,160.345,-54.410,-178.062,6.166,148.536
C01801=1202.176,160.595,-54.431,-178.060,6.167,148.536
C01802=1202.172,160.843,-54.453,-178.057,6.169,148.535
C01803=1202.167,161.092,-54.475,-178.054,6.170,148.535
C01804=1202.162,161.341,-54.497,-178.052,6.172,148.535
C01805=1202.158,161.590,-54.519,-178.049,6.173,148.534
C01806=1202.153,161.840,-54.540,-178.046,6.175,148.534
C01807=1202.148,162.089,-54.562,-178.044,6.176,148.533
C01808=1202.143,162.337,-54.583,-178.041,6.178,148.533
C01809=1202.139,162.587,-54.605,-178.038,6.180,148.533
C01810=1202.134,162.835,-54.627,-178.036,6.181,148.532
C01811=1202.130,163.085,-54.649,-178.033,6.183,148.532
C01812=1202.125,163.333,-54.671,-178.030,6.184,148.531
C01813=1202.120,163.582,-54.692,-178.028,6.186,148.531
C01814=1202.116,163.832,-54.714,-178.026,6.187,148.530
C01815=1202.111,164.081,-54.735,-178.023,6.189,148.530
C01816=1202.106,164.330,-54.757,-178.020,6.191,148.530
C01817=1202.102,164.579,-54.779,-178.018,6.192,148.529
C01818=1202.097,164.828,-54.801,-178.015,6.193,148.529
C01819=1202.092,165.076,-54.823,-178.012,6.195,148.528
C01820=1202.088,165.325,-54.845,-178.010,6.197,148.528
C01821=1202.083,165.574,-54.867,-178.007,6.198,148.528
C01822=1202.078,165.823,-54.888,-178.004,6.200,148.527
C01823=1202.073,166.073,-54.911,-178.002,6.201,148.527
C01824=1202.069,166.321,-54.933,-177.999,6.203,148.527
C01825=1202.064,166.571,-54.955,-177.996,6.204,148.526
C01826=1202.059,166.819,-54.976,-177.994,6.206,148.526
C01827=1202.055,167.069,-54.998,-177.991,6.208,148.525
C01828=1202.050,167.317,-55.020,-177.989,6.209,148.525
C01829=1202.046,167.567,-55.042,-177.986,6.211,148.524
C01830=1202.040,167.816,-55.064,-177.984,6.213,148.524
C01831=1202.036,168.064,-55.087,-177.981,6.214,148.524
C01832=1202.032,168.313,-55.109,-177.978,6.216,148.523
